LIN {X 0,Y 426.46,Z 439.109,A -85,B 0,C 180,E1 20323.799,E2 20323.799} C_VEL
LIN {X 0,Y 426.439,Z 439.071,A -85,B 0,C 180,E1 20319.981,E2 20319.981} C_VEL
LIN {X 0,Y 426.472,Z 439.347,A -85,B 0,C 180,E1 20317.968,E2 20317.968} C_VEL
LIN {X 0,Y 426.886,Z 440.796,A -85,B 0,C 180,E1 20317.446,E2 20317.446} C_VEL
LIN {X 0,Y 428.773,Z 443.794,A -85,B 0,C 180,E1 20316.644,E2 20316.644} C_VEL
LIN {X 0,Y 432.18,Z 446.15,A -85,B 0,C 180,E1 20315.426,E2 20315.426} C_VEL
LIN {X 0,Y 434.235,Z 449.727,A -85,B 0,C 180,E1 20314.641,E2 20314.641} C_VEL
LIN {X 0,Y 437.693,Z 452.592,A -85,B 0,C 180,E1 20313.51,E2 20313.51} C_VEL
LIN {X 0,Y 440.242,Z 456.382,A -85,B 0,C 180,E1 20312.654,E2 20312.654} C_VEL
LIN {X 0,Y 443.022,Z 458.925,A -85,B 0,C 180,E1 20311.818,E2 20311.818} C_VEL
LIN {X 0,Y 446.073,Z 463.006,A -85,B 0,C 180,E1 20310.895,E2 20310.895} C_VEL
LIN {X 0,Y 448.159,Z 465.113,A -85,B 0,C 180,E1 20310.31,E2 20310.31} C_VEL
LIN {X 0,Y 451.831,Z 469.632,A -85,B 0,C 180,E1 20309.293,E2 20309.293} C_VEL
LIN {X 0,Y 458.066,Z 477.379,A -85,B 0,C 180,E1 20307.67,E2 20307.67} C_VEL
LIN {X 0,Y 466.132,Z 487.643,A -85,B 0,C 180,E1 20305.73,E2 20305.73} C_VEL
LIN {X 0,Y 477.609,Z 503.007,A -85,B 0,C 180,E1 20303.219,E2 20303.219} C_VEL
LIN {X 0,Y 488.82,Z 519.176,A -85,B 0,C 180,E1 20300.986,E2 20300.986} C_VEL
LIN {X 0,Y 501.507,Z 538.911,A -85,B 0,C 180,E1 20298.667,E2 20298.667} C_VEL
LIN {X 0,Y 501.955,Z 540.091,A -85,B 0,C 180,E1 20298.578,E2 20298.578} C_VEL
LIN {X 0,Y 490.454,Z 788.265,A -85,B 0,C 180,E1 20294.759,E2 20294.759} C_VEL
LIN {X 0,Y 488.572,Z 820.608,A -85,B 0,C 180,E1 20294.196,E2 20294.196} C_VEL
LIN {X 0,Y 486.489,Z 842.167,A -85,B 0,C 180,E1 20293.667,E2 20293.667} C_VEL
LIN {X 0,Y 483.443,Z 866.539,A -85,B 0,C 180,E1 20292.88,E2 20292.88} C_VEL
LIN {X 0,Y 480.104,Z 887.806,A -85,B 0,C 180,E1 20292.002,E2 20292.002} C_VEL
LIN {X 0,Y 476.07,Z 910.307,A -85,B 0,C 180,E1 20290.877,E2 20290.877} C_VEL
LIN {X 0,Y 471.559,Z 931.55,A -85,B 0,C 180,E1 20289.582,E2 20289.582} C_VEL
LIN {X 0,Y 467.148,Z 950.701,A -85,B 0,C 180,E1 20288.213,E2 20288.213} C_VEL
LIN {X 0,Y 461.702,Z 972.184,A -85,B 0,C 180,E1 20286.398,E2 20286.398} C_VEL
LIN {X 0,Y 457.123,Z 989.065,A -85,B 0,C 180,E1 20284.737,E2 20284.737} C_VEL
LIN {X 0,Y 451.657,Z 1008.264,A -85,B 0,C 180,E1 20282.545,E2 20282.545} C_VEL
LIN {X 0,Y 447.122,Z 1023.569,A -85,B 0,C 180,E1 20280.507,E2 20280.507} C_VEL
LIN {X 0,Y 442.375,Z 1039.686,A -85,B 0,C 180,E1 20278.043,E2 20278.043} C_VEL
LIN {X 0,Y 438.01,Z 1054.252,A -85,B 0,C 180,E1 20275.415,E2 20275.415} C_VEL
LIN {X 0,Y 434.208,Z 1067.674,A -85,B 0,C 180,E1 20272.617,E2 20272.617} C_VEL
LIN {X 0,Y 430.942,Z 1079.536,A -85,B 0,C 180,E1 20269.66,E2 20269.66} C_VEL
LIN {X 0,Y 428.463,Z 1089.76,A -85,B 0,C 180,E1 20266.681,E2 20266.681} C_VEL
LIN {X 0,Y 426.561,Z 1098.496,A -85,B 0,C 180,E1 20263.557,E2 20263.557} C_VEL
LIN {X 0,Y 425.386,Z 1105.117,A -85,B 0,C 180,E1 20260.702,E2 20260.702} C_VEL
LIN {X 0,Y 424.55,Z 1111.253,A -85,B 0,C 180,E1 20257.307,E2 20257.307} C_VEL
LIN {X 0,Y 424.199,Z 1115.035,A -85,B 0,C 180,E1 20254.461,E2 20254.461} C_VEL
LIN {X 0,Y 424.092,Z 1116.75,A -85,B 0,C 180,E1 20252.744,E2 20252.744} C_VEL
LIN {X 0,Y 423.061,Z 1117.653,A -85,B 0,C 180,E1 20251.71,E2 20251.71} C_VEL
LIN {X 0,Y 416.526,Z 1119.369,A -85,B 0,C 180,E1 20248.791,E2 20248.791} C_VEL
LIN {X 0,Y 415.991,Z 1119.509,A -85,B 0,C 180,E1 20248.026,E2 20248.026} C_VEL
LIN {X 0,Y 415.985,Z 1119.493,A -85,B 0,C 180,E1 20245.312,E2 20245.312} C_VEL
LIN {X 0,Y 416.079,Z 1118.241,A -85,B 0,C 180,E1 20242.127,E2 20242.127} C_VEL
LIN {X 0,Y 416.288,Z 1115.397,A -85,B 0,C 180,E1 20238.921,E2 20238.921} C_VEL
LIN {X 0,Y 416.731,Z 1111.601,A -85,B 0,C 180,E1 20235.975,E2 20235.975} C_VEL
LIN {X 0,Y 417.783,Z 1105.394,A -85,B 0,C 180,E1 20232.449,E2 20232.449} C_VEL
LIN {X 0,Y 419.208,Z 1098.674,A -85,B 0,C 180,E1 20229.474,E2 20229.474} C_VEL
LIN {X 0,Y 421.493,Z 1089.722,A -85,B 0,C 180,E1 20226.216,E2 20226.216} C_VEL
LIN {X 0,Y 424.298,Z 1079.776,A -85,B 0,C 180,E1 20223.249,E2 20223.249} C_VEL
LIN {X 0,Y 427.904,Z 1068.257,A -85,B 0,C 180,E1 20220.305,E2 20220.305} C_VEL
LIN {X 0,Y 432.084,Z 1055.296,A -85,B 0,C 180,E1 20217.529,E2 20217.529} C_VEL
LIN {X 0,Y 436.523,Z 1042.037,A -85,B 0,C 180,E1 20215.065,E2 20215.065} C_VEL
LIN {X 0,Y 441.971,Z 1025.703,A -85,B 0,C 180,E1 20212.47,E2 20212.47} C_VEL
LIN {X 0,Y 446.987,Z 1010.498,A -85,B 0,C 180,E1 20210.392,E2 20210.392} C_VEL
LIN {X 0,Y 453.134,Z 991.205,A -85,B 0,C 180,E1 20208.125,E2 20208.125} C_VEL
LIN {X 0,Y 458.273,Z 974.105,A -85,B 0,C 180,E1 20206.412,E2 20206.412} C_VEL
LIN {X 0,Y 463.989,Z 954.018,A -85,B 0,C 180,E1 20204.671,E2 20204.671} C_VEL
LIN {X 0,Y 469.122,Z 933.798,A -85,B 0,C 180,E1 20203.202,E2 20203.202} C_VEL
LIN {X 0,Y 473.862,Z 913.586,A -85,B 0,C 180,E1 20201.952,E2 20201.952} C_VEL
LIN {X 0,Y 478.549,Z 890.327,A -85,B 0,C 180,E1 20200.763,E2 20200.763} C_VEL
LIN {X 0,Y 482.046,Z 870.182,A -85,B 0,C 180,E1 20199.918,E2 20199.918} C_VEL
LIN {X 0,Y 485.569,Z 845.453,A -85,B 0,C 180,E1 20199.092,E2 20199.092} C_VEL
LIN {X 0,Y 487.926,Z 823.544,A -85,B 0,C 180,E1 20198.542,E2 20198.542} C_VEL
LIN {X 0,Y 489.763,Z 798.161,A -85,B 0,C 180,E1 20198.071,E2 20198.071} C_VEL
LIN {X 0,Y 502.56,Z 550.013,A -85,B 0,C 180,E1 20194.222,E2 20194.222} C_VEL
LIN {X 0,Y 502.637,Z 546.862,A -85,B 0,C 180,E1 20194.158,E2 20194.158} C_VEL
LIN {X 0,Y 491.988,Z 530.606,A -85,B 0,C 180,E1 20191.967,E2 20191.967} C_VEL
LIN {X 0,Y 481.908,Z 516.077,A -85,B 0,C 180,E1 20189.695,E2 20189.695} C_VEL
LIN {X 0,Y 470.549,Z 500.825,A -85,B 0,C 180,E1 20186.843,E2 20186.843} C_VEL
LIN {X 0,Y 464.667,Z 493.605,A -85,B 0,C 180,E1 20185.218,E2 20185.218} C_VEL
LIN {X 0,Y 461.386,Z 489.465,A -85,B 0,C 180,E1 20184.247,E2 20184.247} C_VEL
LIN {X 0,Y 456.943,Z 483.981,A -85,B 0,C 180,E1 20182.856,E2 20182.856} C_VEL
LIN {X 0,Y 453.182,Z 479.216,A -85,B 0,C 180,E1 20181.587,E2 20181.587} C_VEL
LIN {X 0,Y 449.14,Z 474.869,A -85,B 0,C 180,E1 20180.152,E2 20180.152} C_VEL
LIN {X 0,Y 447.664,Z 472.755,A -85,B 0,C 180,E1 20179.575,E2 20179.575} C_VEL
LIN {X 0,Y 444.246,Z 469.377,A -85,B 0,C 180,E1 20178.232,E2 20178.232} C_VEL
LIN {X 0,Y 442.58,Z 466.748,A -85,B 0,C 180,E1 20177.486,E2 20177.486} C_VEL
LIN {X 0,Y 439.326,Z 464.015,A -85,B 0,C 180,E1 20176.053,E2 20176.053} C_VEL
LIN {X 0,Y 437.017,Z 460.34,A -85,B 0,C 180,E1 20174.848,E2 20174.848} C_VEL
LIN {X 0,Y 433.502,Z 457.818,A -85,B 0,C 180,E1 20172.996,E2 20172.996} C_VEL
LIN {X 0,Y 431.27,Z 453.931,A -85,B 0,C 180,E1 20171.501,E2 20171.501} C_VEL
LIN {X 0,Y 427.253,Z 451.254,A -85,B 0,C 180,E1 20168.614,E2 20168.614} C_VEL
LIN {X 0,Y 425.405,Z 447.905,A -85,B 0,C 180,E1 20166.681,E2 20166.681} C_VEL
LIN {X 0,Y 424.103,Z 446.752,A -85,B 0,C 180,E1 20165.14,E2 20165.14} C_VEL
LIN {X 0,Y 421.605,Z 445.43,A -85,B 0,C 180,E1 20158.777,E2 20158.777} C_VEL
LIN {X 0,Y 423.828,Z 446.628,A -85,B 0,C 180,E1 20152.681,E2 20152.681} C_VEL
LIN {X 0,Y 425.295,Z 447.708,A -85,B 0,C 180,E1 20150.912,E2 20150.912} C_VEL
LIN {X 0,Y 427.312,Z 451.295,A -85,B 0,C 180,E1 20148.801,E2 20148.801} C_VEL
LIN {X 0,Y 431.535,Z 454.284,A -85,B 0,C 180,E1 20145.782,E2 20145.782} C_VEL
LIN {X 0,Y 433.596,Z 457.858,A -85,B 0,C 180,E1 20144.416,E2 20144.416} C_VEL
LIN {X 0,Y 437.41,Z 460.857,A -85,B 0,C 180,E1 20142.409,E2 20142.409} C_VEL
LIN {X 0,Y 439.838,Z 464.601,A -85,B 0,C 180,E1 20141.167,E2 20141.167} C_VEL
LIN {X 0,Y 442.831,Z 467.253,A -85,B 0,C 180,E1 20139.859,E2 20139.859} C_VEL
LIN {X 0,Y 448.06,Z 474.081,A -85,B 0,C 180,E1 20137.705,E2 20137.705} C_VEL
LIN {X 0,Y 451.148,Z 477.881,A -85,B 0,C 180,E1 20136.557,E2 20136.557} C_VEL
LIN {X 0,Y 456.118,Z 484.462,A -85,B 0,C 180,E1 20134.831,E2 20134.831} C_VEL
LIN {X 0,Y 462.851,Z 493.629,A -85,B 0,C 180,E1 20132.708,E2 20132.708} C_VEL
LIN {X 0,Y 470.507,Z 504.351,A -85,B 0,C 180,E1 20130.53,E2 20130.53} C_VEL
LIN {X 0,Y 479.766,Z 518.204,A -85,B 0,C 180,E1 20128.143,E2 20128.143} C_VEL
LIN {X 0,Y 489.997,Z 534.394,A -85,B 0,C 180,E1 20125.757,E2 20125.757} C_VEL
LIN {X 0,Y 500.548,Z 552.647,A -85,B 0,C 180,E1 20123.503,E2 20123.503} C_VEL
LIN {X 0,Y 502.46,Z 556.456,A -85,B 0,C 180,E1 20123.105,E2 20123.105} C_VEL
LIN {X 0,Y 491.286,Z 774.343,A -85,B 0,C 180,E1 20119.712,E2 20119.712} C_VEL
LIN {X 0,Y 487.957,Z 837.015,A -85,B 0,C 180,E1 20118.712,E2 20118.712} C_VEL
LIN {X 0,Y 485.355,Z 862.027,A -85,B 0,C 180,E1 20118.161,E2 20118.161} C_VEL
LIN {X 0,Y 482.318,Z 883.724,A -85,B 0,C 180,E1 20117.534,E2 20117.534} C_VEL
LIN {X 0,Y 478.102,Z 908.208,A -85,B 0,C 180,E1 20116.615,E2 20116.615} C_VEL
LIN {X 0,Y 473.961,Z 928.701,A -85,B 0,C 180,E1 20115.657,E2 20115.657} C_VEL
LIN {X 0,Y 468.64,Z 952.137,A -85,B 0,C 180,E1 20114.327,E2 20114.327} C_VEL
LIN {X 0,Y 463.55,Z 971.992,A -85,B 0,C 180,E1 20112.971,E2 20112.971} C_VEL
LIN {X 0,Y 457.782,Z 993.134,A -85,B 0,C 180,E1 20111.272,E2 20111.272} C_VEL
LIN {X 0,Y 452.241,Z 1011.721,A -85,B 0,C 180,E1 20109.499,E2 20109.499} C_VEL
LIN {X 0,Y 446.85,Z 1029.266,A -85,B 0,C 180,E1 20107.572,E2 20107.572} C_VEL
LIN {X 0,Y 440.903,Z 1047.883,A -85,B 0,C 180,E1 20105.172,E2 20105.172} C_VEL
LIN {X 0,Y 436.087,Z 1062.963,A -85,B 0,C 180,E1 20102.916,E2 20102.916} C_VEL
LIN {X 0,Y 430.911,Z 1079.333,A -85,B 0,C 180,E1 20100.058,E2 20100.058} C_VEL
LIN {X 0,Y 427.044,Z 1092.048,A -85,B 0,C 180,E1 20097.469,E2 20097.469} C_VEL
LIN {X 0,Y 423.093,Z 1105.982,A -85,B 0,C 180,E1 20094.133,E2 20094.133} C_VEL
LIN {X 0,Y 420.586,Z 1115.872,A -85,B 0,C 180,E1 20091.33,E2 20091.33} C_VEL
LIN {X 0,Y 418.345,Z 1126.251,A -85,B 0,C 180,E1 20087.814,E2 20087.814} C_VEL
LIN {X 0,Y 417.128,Z 1133.344,A -85,B 0,C 180,E1 20084.862,E2 20084.862} C_VEL
LIN {X 0,Y 416.363,Z 1139.65,A -85,B 0,C 180,E1 20081.638,E2 20081.638} C_VEL
LIN {X 0,Y 416.046,Z 1144.213,A -85,B 0,C 180,E1 20078.43,E2 20078.43} C_VEL
LIN {X 0,Y 415.959,Z 1147.017,A -85,B 0,C 180,E1 20075.656,E2 20075.656} C_VEL
LIN {X 0,Y 415.968,Z 1148.924,A -85,B 0,C 180,E1 20072.48,E2 20072.48} C_VEL
LIN {X 0,Y 415.979,Z 1149.195,A -85,B 0,C 180,E1 20069.404,E2 20069.404} C_VEL
LIN {X 0,Y 415.969,Z 1148.403,A -85,B 0,C 180,E1 20066.831,E2 20066.831} C_VEL
LIN {X 0,Y 415.973,Z 1146.597,A -85,B 0,C 180,E1 20064.206,E2 20064.206} C_VEL
LIN {X 0,Y 416.069,Z 1143.094,A -85,B 0,C 180,E1 20061.01,E2 20061.01} C_VEL
LIN {X 0,Y 416.452,Z 1137.87,A -85,B 0,C 180,E1 20057.802,E2 20057.802} C_VEL
LIN {X 0,Y 417.143,Z 1132.089,A -85,B 0,C 180,E1 20054.997,E2 20054.997} C_VEL
LIN {X 0,Y 418.646,Z 1123.03,A -85,B 0,C 180,E1 20051.477,E2 20051.477} C_VEL
LIN {X 0,Y 420.46,Z 1114.223,A -85,B 0,C 180,E1 20048.663,E2 20048.663} C_VEL
LIN {X 0,Y 423.336,Z 1102.294,A -85,B 0,C 180,E1 20045.436,E2 20045.436} C_VEL
LIN {X 0,Y 426.568,Z 1090.052,A -85,B 0,C 180,E1 20042.649,E2 20042.649} C_VEL
LIN {X 0,Y 430.565,Z 1076.099,A -85,B 0,C 180,E1 20039.893,E2 20039.893} C_VEL
LIN {X 0,Y 435.182,Z 1060.223,A -85,B 0,C 180,E1 20037.24,E2 20037.24} C_VEL
LIN {X 0,Y 440.295,Z 1043.196,A -85,B 0,C 180,E1 20034.772,E2 20034.772} C_VEL
LIN {X 0,Y 445.372,Z 1025.808,A -85,B 0,C 180,E1 20032.632,E2 20032.632} C_VEL
LIN {X 0,Y 450.584,Z 1007.658,A -85,B 0,C 180,E1 20030.687,E2 20030.687} C_VEL
LIN {X 0,Y 456.176,Z 986.891,A -85,B 0,C 180,E1 20028.802,E2 20028.802} C_VEL
LIN {X 0,Y 460.927,Z 968.157,A -85,B 0,C 180,E1 20027.341,E2 20027.341} C_VEL
LIN {X 0,Y 466.322,Z 944.965,A -85,B 0,C 180,E1 20025.824,E2 20025.824} C_VEL
LIN {X 0,Y 470.495,Z 924.844,A -85,B 0,C 180,E1 20024.724,E2 20024.724} C_VEL
LIN {X 0,Y 475.036,Z 899.834,A -85,B 0,C 180,E1 20023.608,E2 20023.608} C_VEL
LIN {X 0,Y 478.393,Z 877.83,A -85,B 0,C 180,E1 20022.836,E2 20022.836} C_VEL
LIN {X 0,Y 481.549,Z 851.869,A -85,B 0,C 180,E1 20022.143,E2 20022.143} C_VEL
LIN {X 0,Y 483.347,Z 829.268,A -85,B 0,C 180,E1 20021.7,E2 20021.7} C_VEL
LIN {X 0,Y 493.938,Z 604.352,A -85,B 0,C 180,E1 20018.193,E2 20018.193} C_VEL
LIN {X 0,Y 496.302,Z 552.568,A -85,B 0,C 180,E1 20017.368,E2 20017.368} C_VEL
LIN {X 0,Y 485.264,Z 532.833,A -85,B 0,C 180,E1 20015.254,E2 20015.254} C_VEL
LIN {X 0,Y 475.654,Z 517.03,A -85,B 0,C 180,E1 20013.275,E2 20013.275} C_VEL
LIN {X 0,Y 465.604,Z 501.38,A -85,B 0,C 180,E1 20011.025,E2 20011.025} C_VEL
LIN {X 0,Y 456.759,Z 488.546,A -85,B 0,C 180,E1 20008.862,E2 20008.862} C_VEL
LIN {X 0,Y 446.922,Z 474.863,A -85,B 0,C 180,E1 20006.187,E2 20006.187} C_VEL
LIN {X 0,Y 441.259,Z 467.655,A -85,B 0,C 180,E1 20004.499,E2 20004.499} C_VEL
LIN {X 0,Y 434.601,Z 459.158,A -85,B 0,C 180,E1 20002.31,E2 20002.31} C_VEL
LIN {X 0,Y 431.388,Z 455.946,A -85,B 0,C 180,E1 20001.198,E2 20001.198} C_VEL
LIN {X 0,Y 429.776,Z 453.269,A -85,B 0,C 180,E1 20000.567,E2 20000.567} C_VEL
LIN {X 0,Y 426.394,Z 450.626,A -85,B 0,C 180,E1 19999.308,E2 19999.308} C_VEL
LIN {X 0,Y 424.043,Z 446.767,A -85,B 0,C 180,E1 19998.277,E2 19998.277} C_VEL
LIN {X 0,Y 420.526,Z 444.455,A -85,B 0,C 180,E1 19996.792,E2 19996.792} C_VEL
LIN {X 0,Y 418.726,Z 441.079,A -85,B 0,C 180,E1 19995.774,E2 19995.774} C_VEL
LIN {X 0,Y 418.542,Z 440.13,A -85,B 0,C 180,E1 19995.094,E2 19995.094} C_VEL
LIN {X 0,Y 418.532,Z 440.092,A -85,B 0,C 180,E1 19991.158,E2 19991.158} C_VEL
LIN {X 0,Y 418.538,Z 440.058,A -85,B 0,C 180,E1 19987.274,E2 19987.274} C_VEL
LIN {X 0,Y 418.532,Z 440.043,A -85,B 0,C 180,E1 19983.424,E2 19983.424} C_VEL
LIN {X 0,Y 418.546,Z 440.076,A -85,B 0,C 180,E1 19979.589,E2 19979.589} C_VEL
LIN {X 0,Y 418.537,Z 440.068,A -85,B 0,C 180,E1 19975.616,E2 19975.616} C_VEL
LIN {X 0,Y 418.535,Z 440.041,A -85,B 0,C 180,E1 19971.759,E2 19971.759} C_VEL
LIN {X 0,Y 418.514,Z 440.068,A -85,B 0,C 180,E1 19968.003,E2 19968.003} C_VEL
LIN {X 0,Y 418.501,Z 440.084,A -85,B 0,C 180,E1 19964.194,E2 19964.194} C_VEL
LIN {X 0,Y 418.566,Z 440.34,A -85,B 0,C 180,E1 19961.083,E2 19961.083} C_VEL
LIN {X 0,Y 418.885,Z 441.719,A -85,B 0,C 180,E1 19960.517,E2 19960.517} C_VEL
LIN {X 0,Y 420.634,Z 444.556,A -85,B 0,C 180,E1 19959.62,E2 19959.62} C_VEL
LIN {X 0,Y 424.541,Z 447.376,A -85,B 0,C 180,E1 19957.971,E2 19957.971} C_VEL
LIN {X 0,Y 426.527,Z 450.821,A -85,B 0,C 180,E1 19957.098,E2 19957.098} C_VEL
LIN {X 0,Y 429.581,Z 453.153,A -85,B 0,C 180,E1 19955.963,E2 19955.963} C_VEL
LIN {X 0,Y 430.325,Z 454.138,A -85,B 0,C 180,E1 19955.679,E2 19955.679} C_VEL
LIN {X 0,Y 432.755,Z 457.679,A -85,B 0,C 180,E1 19954.767,E2 19954.767} C_VEL
LIN {X 0,Y 435.613,Z 460.182,A -85,B 0,C 180,E1 19953.814,E2 19953.814} C_VEL
LIN {X 0,Y 438.633,Z 464.237,A -85,B 0,C 180,E1 19952.803,E2 19952.803} C_VEL
LIN {X 0,Y 440.788,Z 466.318,A -85,B 0,C 180,E1 19952.141,E2 19952.141} C_VEL
LIN {X 0,Y 444.326,Z 470.77,A -85,B 0,C 180,E1 19951.064,E2 19951.064} C_VEL
LIN {X 0,Y 446.059,Z 472.796,A -85,B 0,C 180,E1 19950.562,E2 19950.562} C_VEL
LIN {X 0,Y 450.981,Z 478.829,A -85,B 0,C 180,E1 19949.192,E2 19949.192} C_VEL
LIN {X 0,Y 456.103,Z 485.324,A -85,B 0,C 180,E1 19947.848,E2 19947.848} C_VEL
LIN {X 0,Y 463.181,Z 494.394,A -85,B 0,C 180,E1 19946.117,E2 19946.117} C_VEL
LIN {X 0,Y 474.648,Z 509.946,A -85,B 0,C 180,E1 19943.554,E2 19943.554} C_VEL
LIN {X 0,Y 485.547,Z 525.916,A -85,B 0,C 180,E1 19941.336,E2 19941.336} C_VEL
LIN {X 0,Y 496.73,Z 543.494,A -85,B 0,C 180,E1 19939.24,E2 19939.24} C_VEL
LIN {X 0,Y 484.803,Z 792.502,A -85,B 0,C 180,E1 19935.383,E2 19935.383} C_VEL
LIN {X 0,Y 482.96,Z 821.822,A -85,B 0,C 180,E1 19934.857,E2 19934.857} C_VEL
LIN {X 0,Y 480.821,Z 843.2,A -85,B 0,C 180,E1 19934.325,E2 19934.325} C_VEL
LIN {X 0,Y 477.432,Z 868.992,A -85,B 0,C 180,E1 19933.471,E2 19933.471} C_VEL
LIN {X 0,Y 474.057,Z 889.712,A -85,B 0,C 180,E1 19932.598,E2 19932.598} C_VEL
LIN {X 0,Y 469.603,Z 913.272,A -85,B 0,C 180,E1 19931.386,E2 19931.386} C_VEL
LIN {X 0,Y 465.228,Z 933.159,A -85,B 0,C 180,E1 19930.149,E2 19930.149} C_VEL
LIN {X 0,Y 460.321,Z 953.773,A -85,B 0,C 180,E1 19928.645,E2 19928.645} C_VEL
LIN {X 0,Y 455.08,Z 973.456,A -85,B 0,C 180,E1 19926.937,E2 19926.937} C_VEL
LIN {X 0,Y 450.365,Z 990.25,A -85,B 0,C 180,E1 19925.257,E2 19925.257} C_VEL
LIN {X 0,Y 444.542,Z 1009.868,A -85,B 0,C 180,E1 19922.968,E2 19922.968} C_VEL
LIN {X 0,Y 439.898,Z 1024.996,A -85,B 0,C 180,E1 19920.911,E2 19920.911} C_VEL
LIN {X 0,Y 434.659,Z 1041.964,A -85,B 0,C 180,E1 19918.23,E2 19918.23} C_VEL
LIN {X 0,Y 430.493,Z 1055.403,A -85,B 0,C 180,E1 19915.743,E2 19915.743} C_VEL
LIN {X 0,Y 426.386,Z 1069.23,A -85,B 0,C 180,E1 19912.764,E2 19912.764} C_VEL
LIN {X 0,Y 423.316,Z 1079.957,A -85,B 0,C 180,E1 19910.029,E2 19910.029} C_VEL
LIN {X 0,Y 420.717,Z 1090.164,A -85,B 0,C 180,E1 19906.997,E2 19906.997} C_VEL
LIN {X 0,Y 418.715,Z 1098.875,A -85,B 0,C 180,E1 19903.816,E2 19903.816} C_VEL
LIN {X 0,Y 417.466,Z 1105.533,A -85,B 0,C 180,E1 19900.884,E2 19900.884} C_VEL
LIN {X 0,Y 416.586,Z 1111.593,A -85,B 0,C 180,E1 19897.447,E2 19897.447} C_VEL
LIN {X 0,Y 416.216,Z 1115.361,A -85,B 0,C 180,E1 19894.547,E2 19894.547} C_VEL
LIN {X 0,Y 416.027,Z 1118.287,A -85,B 0,C 180,E1 19891.239,E2 19891.239} C_VEL
LIN {X 0,Y 415.991,Z 1119.502,A -85,B 0,C 180,E1 19888.072,E2 19888.072} C_VEL
LIN {X 0,Y 415.991,Z 1119.509,A -85,B 0,C 180,E1 19888.026,E2 19888.026} C_VEL
LIN {X 0,Y 415.009,Z 1119.736,A -85,B 0,C 180,E1 19886.965,E2 19886.965} C_VEL
LIN {X 0,Y 408.577,Z 1119.451,A -85,B 0,C 180,E1 19883.975,E2 19883.975} C_VEL
LIN {X 0,Y 408.034,Z 1119.09,A -85,B 0,C 180,E1 19883.196,E2 19883.196} C_VEL
LIN {X 0,Y 408.156,Z 1117.287,A -85,B 0,C 180,E1 19880.411,E2 19880.411} C_VEL
LIN {X 0,Y 408.589,Z 1113.451,A -85,B 0,C 180,E1 19876.845,E2 19876.845} C_VEL
LIN {X 0,Y 409.323,Z 1108.812,A -85,B 0,C 180,E1 19873.831,E2 19873.831} C_VEL
LIN {X 0,Y 410.725,Z 1102.108,A -85,B 0,C 180,E1 19870.414,E2 19870.414} C_VEL
LIN {X 0,Y 412.729,Z 1093.989,A -85,B 0,C 180,E1 19867.193,E2 19867.193} C_VEL
LIN {X 0,Y 415.366,Z 1084.91,A -85,B 0,C 180,E1 19864.169,E2 19864.169} C_VEL
LIN {X 0,Y 418.955,Z 1073.52,A -85,B 0,C 180,E1 19861.021,E2 19861.021} C_VEL
LIN {X 0,Y 422.775,Z 1062.109,A -85,B 0,C 180,E1 19858.329,E2 19858.329} C_VEL
LIN {X 0,Y 428.108,Z 1046.738,A -85,B 0,C 180,E1 19855.257,E2 19855.257} C_VEL
LIN {X 0,Y 432.884,Z 1033.061,A -85,B 0,C 180,E1 19852.924,E2 19852.924} C_VEL
LIN {X 0,Y 438.969,Z 1015.438,A -85,B 0,C 180,E1 19850.345,E2 19850.345} C_VEL
LIN {X 0,Y 444.337,Z 999.378,A -85,B 0,C 180,E1 19848.34,E2 19848.34} C_VEL
LIN {X 0,Y 450.441,Z 980.418,A -85,B 0,C 180,E1 19846.297,E2 19846.297} C_VEL
LIN {X 0,Y 455.879,Z 962.101,A -85,B 0,C 180,E1 19844.624,E2 19844.624} C_VEL
LIN {X 0,Y 461.101,Z 943.313,A -85,B 0,C 180,E1 19843.139,E2 19843.139} C_VEL
LIN {X 0,Y 466.575,Z 921.361,A -85,B 0,C 180,E1 19841.681,E2 19841.681} C_VEL
LIN {X 0,Y 470.861,Z 902.128,A -85,B 0,C 180,E1 19840.609,E2 19840.609} C_VEL
LIN {X 0,Y 475.391,Z 878.698,A -85,B 0,C 180,E1 19839.521,E2 19839.521} C_VEL
LIN {X 0,Y 478.772,Z 857.301,A -85,B 0,C 180,E1 19838.73,E2 19838.73} C_VEL
LIN {X 0,Y 481.845,Z 833.683,A -85,B 0,C 180,E1 19838.04,E2 19838.04} C_VEL
LIN {X 0,Y 483.974,Z 809.348,A -85,B 0,C 180,E1 19837.53,E2 19837.53} C_VEL
LIN {X 0,Y 496.518,Z 575.381,A -85,B 0,C 180,E1 19833.865,E2 19833.865} C_VEL
LIN {X 0,Y 497.779,Z 550.89,A -85,B 0,C 180,E1 19833.469,E2 19833.469} C_VEL
LIN {X 0,Y 486.39,Z 533.438,A -85,B 0,C 180,E1 19831.029,E2 19831.029} C_VEL
LIN {X 0,Y 477.111,Z 520.336,A -85,B 0,C 180,E1 19828.852,E2 19828.852} C_VEL
LIN {X 0,Y 467.91,Z 507.726,A -85,B 0,C 180,E1 19826.459,E2 19826.459} C_VEL
LIN {X 0,Y 459.463,Z 497.013,A -85,B 0,C 180,E1 19824.014,E2 19824.014} C_VEL
LIN {X 0,Y 454.702,Z 491.162,A -85,B 0,C 180,E1 19822.497,E2 19822.497} C_VEL
LIN {X 0,Y 450.397,Z 485.874,A -85,B 0,C 180,E1 19821.01,E2 19821.01} C_VEL
LIN {X 0,Y 446.739,Z 481.525,A -85,B 0,C 180,E1 19819.651,E2 19819.651} C_VEL
LIN {X 0,Y 445.574,Z 480.089,A -85,B 0,C 180,E1 19819.193,E2 19819.193} C_VEL
LIN {X 0,Y 442.111,Z 476.312,A -85,B 0,C 180,E1 19817.778,E2 19817.778} C_VEL
LIN {X 0,Y 440.736,Z 474.286,A -85,B 0,C 180,E1 19817.153,E2 19817.153} C_VEL
LIN {X 0,Y 437.441,Z 471.214,A -85,B 0,C 180,E1 19815.648,E2 19815.648} C_VEL
LIN {X 0,Y 435.543,Z 468.086,A -85,B 0,C 180,E1 19814.627,E2 19814.627} C_VEL
LIN {X 0,Y 432.091,Z 465.501,A -85,B 0,C 180,E1 19812.768,E2 19812.768} C_VEL
LIN {X 0,Y 429.898,Z 461.671,A -85,B 0,C 180,E1 19811.267,E2 19811.267} C_VEL
LIN {X 0,Y 426.124,Z 459.141,A -85,B 0,C 180,E1 19808.501,E2 19808.501} C_VEL
LIN {X 0,Y 424.242,Z 455.75,A -85,B 0,C 180,E1 19806.496,E2 19806.496} C_VEL
LIN {X 0,Y 423.024,Z 454.66,A -85,B 0,C 180,E1 19805.017,E2 19805.017} C_VEL
LIN {X 0,Y 420.63,Z 453.371,A -85,B 0,C 180,E1 19798.774,E2 19798.774} C_VEL
LIN {X 0,Y 422.86,Z 454.575,A -85,B 0,C 180,E1 19792.664,E2 19792.664} C_VEL
LIN {X 0,Y 424.236,Z 455.676,A -85,B 0,C 180,E1 19790.983,E2 19790.983} C_VEL
LIN {X 0,Y 426.039,Z 459.015,A -85,B 0,C 180,E1 19789.041,E2 19789.041} C_VEL
LIN {X 0,Y 429.781,Z 461.587,A -85,B 0,C 180,E1 19786.272,E2 19786.272} C_VEL
LIN {X 0,Y 432.63,Z 466.024,A -85,B 0,C 180,E1 19784.38,E2 19784.38} C_VEL
LIN {X 0,Y 435.825,Z 468.515,A -85,B 0,C 180,E1 19782.682,E2 19782.682} C_VEL
LIN {X 0,Y 438.474,Z 472.437,A -85,B 0,C 180,E1 19781.313,E2 19781.313} C_VEL
LIN {X 0,Y 441.286,Z 475.021,A -85,B 0,C 180,E1 19780.061,E2 19780.061} C_VEL
LIN {X 0,Y 448.943,Z 484.904,A -85,B 0,C 180,E1 19776.956,E2 19776.956} C_VEL
LIN {X 0,Y 454.156,Z 491.981,A -85,B 0,C 180,E1 19775.102,E2 19775.102} C_VEL
LIN {X 0,Y 460.626,Z 500.936,A -85,B 0,C 180,E1 19773.02,E2 19773.02} C_VEL
LIN {X 0,Y 468.796,Z 512.579,A -85,B 0,C 180,E1 19770.657,E2 19770.657} C_VEL
LIN {X 0,Y 479.429,Z 528.801,A -85,B 0,C 180,E1 19767.906,E2 19767.906} C_VEL
LIN {X 0,Y 489.486,Z 545.494,A -85,B 0,C 180,E1 19765.557,E2 19765.557} C_VEL
LIN {X 0,Y 497.614,Z 560.041,A -85,B 0,C 180,E1 19763.799,E2 19763.799} C_VEL
LIN {X 0,Y 486.071,Z 777.932,A -85,B 0,C 180,E1 19760.388,E2 19760.388} C_VEL
LIN {X 0,Y 482.807,Z 837.069,A -85,B 0,C 180,E1 19759.438,E2 19759.438} C_VEL
LIN {X 0,Y 480.136,Z 861.939,A -85,B 0,C 180,E1 19758.886,E2 19758.886} C_VEL
LIN {X 0,Y 476.977,Z 883.884,A -85,B 0,C 180,E1 19758.249,E2 19758.249} C_VEL
LIN {X 0,Y 472.616,Z 908.39,A -85,B 0,C 180,E1 19757.324,E2 19757.324} C_VEL
LIN {X 0,Y 468.36,Z 928.824,A -85,B 0,C 180,E1 19756.363,E2 19756.363} C_VEL
LIN {X 0,Y 462.878,Z 952.174,A -85,B 0,C 180,E1 19755.028,E2 19755.028} C_VEL
LIN {X 0,Y 457.728,Z 971.632,A -85,B 0,C 180,E1 19753.692,E2 19753.692} C_VEL
LIN {X 0,Y 451.88,Z 992.414,A -85,B 0,C 180,E1 19752.017,E2 19752.017} C_VEL
LIN {X 0,Y 445.875,Z 1011.878,A -85,B 0,C 180,E1 19750.146,E2 19750.146} C_VEL
LIN {X 0,Y 440.188,Z 1029.73,A -85,B 0,C 180,E1 19748.16,E2 19748.16} C_VEL
LIN {X 0,Y 434.184,Z 1047.755,A -85,B 0,C 180,E1 19745.799,E2 19745.799} C_VEL
LIN {X 0,Y 428.887,Z 1063.669,A -85,B 0,C 180,E1 19743.381,E2 19743.381} C_VEL
LIN {X 0,Y 423.793,Z 1079.06,A -85,B 0,C 180,E1 19740.639,E2 19740.639} C_VEL
LIN {X 0,Y 419.702,Z 1091.864,A -85,B 0,C 180,E1 19737.991,E2 19737.991} C_VEL
LIN {X 0,Y 415.551,Z 1105.776,A -85,B 0,C 180,E1 19734.599,E2 19734.599} C_VEL
LIN {X 0,Y 412.899,Z 1115.656,A -85,B 0,C 180,E1 19731.747,E2 19731.747} C_VEL
LIN {X 0,Y 410.521,Z 1126.017,A -85,B 0,C 180,E1 19728.166,E2 19728.166} C_VEL
LIN {X 0,Y 409.223,Z 1133.103,A -85,B 0,C 180,E1 19725.156,E2 19725.156} C_VEL
LIN {X 0,Y 408.398,Z 1139.396,A -85,B 0,C 180,E1 19721.868,E2 19721.868} C_VEL
LIN {X 0,Y 408.054,Z 1143.95,A -85,B 0,C 180,E1 19718.596,E2 19718.596} C_VEL
LIN {X 0,Y 407.966,Z 1146.749,A -85,B 0,C 180,E1 19715.767,E2 19715.767} C_VEL
LIN {X 0,Y 407.971,Z 1148.645,A -85,B 0,C 180,E1 19712.528,E2 19712.528} C_VEL
LIN {X 0,Y 407.985,Z 1148.898,A -85,B 0,C 180,E1 19709.337,E2 19709.337} C_VEL
LIN {X 0,Y 407.978,Z 1148.037,A -85,B 0,C 180,E1 19706.628,E2 19706.628} C_VEL
LIN {X 0,Y 407.988,Z 1145.942,A -85,B 0,C 180,E1 19703.668,E2 19703.668} C_VEL
LIN {X 0,Y 408.136,Z 1141.932,A -85,B 0,C 180,E1 19700.268,E2 19700.268} C_VEL
LIN {X 0,Y 408.558,Z 1137.015,A -85,B 0,C 180,E1 19697.275,E2 19697.275} C_VEL
LIN {X 0,Y 409.502,Z 1130.174,A -85,B 0,C 180,E1 19693.983,E2 19693.983} C_VEL
LIN {X 0,Y 411.085,Z 1121.426,A -85,B 0,C 180,E1 19690.683,E2 19690.683} C_VEL
LIN {X 0,Y 413.333,Z 1111.496,A -85,B 0,C 180,E1 19687.529,E2 19687.529} C_VEL
LIN {X 0,Y 416.4,Z 1099.549,A -85,B 0,C 180,E1 19684.391,E2 19684.391} C_VEL
LIN {X 0,Y 419.972,Z 1087.045,A -85,B 0,C 180,E1 19681.564,E2 19681.564} C_VEL
LIN {X 0,Y 424.299,Z 1072.517,A -85,B 0,C 180,E1 19678.772,E2 19678.772} C_VEL
LIN {X 0,Y 428.753,Z 1058.04,A -85,B 0,C 180,E1 19676.363,E2 19676.363} C_VEL
LIN {X 0,Y 434.459,Z 1039.619,A -85,B 0,C 180,E1 19673.738,E2 19673.738} C_VEL
LIN {X 0,Y 439.377,Z 1023.431,A -85,B 0,C 180,E1 19671.757,E2 19671.757} C_VEL
LIN {X 0,Y 445.321,Z 1003.183,A -85,B 0,C 180,E1 19669.626,E2 19669.626} C_VEL
LIN {X 0,Y 450.402,Z 984.835,A -85,B 0,C 180,E1 19667.984,E2 19667.984} C_VEL
LIN {X 0,Y 455.874,Z 963.878,A -85,B 0,C 180,E1 19666.37,E2 19666.37} C_VEL
LIN {X 0,Y 460.94,Z 942.268,A -85,B 0,C 180,E1 19664.994,E2 19664.994} C_VEL
LIN {X 0,Y 465.595,Z 920.305,A -85,B 0,C 180,E1 19663.815,E2 19663.815} C_VEL
LIN {X 0,Y 469.713,Z 897.509,A -85,B 0,C 180,E1 19662.832,E2 19662.832} C_VEL
LIN {X 0,Y 473.087,Z 875.77,A -85,B 0,C 180,E1 19662.08,E2 19662.08} C_VEL
LIN {X 0,Y 476.23,Z 849.82,A -85,B 0,C 180,E1 19661.403,E2 19661.403} C_VEL
LIN {X 0,Y 478.004,Z 827.39,A -85,B 0,C 180,E1 19660.968,E2 19660.968} C_VEL
LIN {X 0,Y 488.95,Z 602.172,A -85,B 0,C 180,E1 19657.436,E2 19657.436} C_VEL
LIN {X 0,Y 491.115,Z 556.093,A -85,B 0,C 180,E1 19656.695,E2 19656.695} C_VEL
LIN {X 0,Y 480.584,Z 537.168,A -85,B 0,C 180,E1 19654.611,E2 19654.611} C_VEL
LIN {X 0,Y 469.777,Z 519.215,A -85,B 0,C 180,E1 19652.292,E2 19652.292} C_VEL
LIN {X 0,Y 458.2,Z 501.404,A -85,B 0,C 180,E1 19649.55,E2 19649.55} C_VEL
LIN {X 0,Y 447.654,Z 486.414,A -85,B 0,C 180,E1 19646.749,E2 19646.749} C_VEL
LIN {X 0,Y 442.891,Z 480.104,A -85,B 0,C 180,E1 19645.365,E2 19645.365} C_VEL
LIN {X 0,Y 439.123,Z 475.014,A -85,B 0,C 180,E1 19644.196,E2 19644.196} C_VEL
LIN {X 0,Y 432.547,Z 466.571,A -85,B 0,C 180,E1 19641.993,E2 19641.993} C_VEL
LIN {X 0,Y 429.22,Z 463.073,A -85,B 0,C 180,E1 19640.809,E2 19640.809} C_VEL
LIN {X 0,Y 427.784,Z 460.77,A -85,B 0,C 180,E1 19640.239,E2 19640.239} C_VEL
LIN {X 0,Y 424.474,Z 457.977,A -85,B 0,C 180,E1 19638.97,E2 19638.97} C_VEL
LIN {X 0,Y 422.46,Z 454.5,A -85,B 0,C 180,E1 19638.063,E2 19638.063} C_VEL
LIN {X 0,Y 418.99,Z 452.142,A -85,B 0,C 180,E1 19636.57,E2 19636.57} C_VEL
LIN {X 0,Y 417.008,Z 448.893,A -85,B 0,C 180,E1 19635.542,E2 19635.542} C_VEL
LIN {X 0,Y 416.049,Z 447.727,A -85,B 0,C 180,E1 19635.044,E2 19635.044} C_VEL
LIN {X 0,Y 412.517,Z 445.326,A -85,B 0,C 180,E1 19633.17,E2 19633.17} C_VEL
LIN {X 0,Y 410.736,Z 441.861,A -85,B 0,C 180,E1 19631.8,E2 19631.8} C_VEL
LIN {X 0,Y 410.594,Z 441.11,A -85,B 0,C 180,E1 19630.808,E2 19630.808} C_VEL
LIN {X 0,Y 410.583,Z 441.057,A -85,B 0,C 180,E1 19626.853,E2 19626.853} C_VEL
LIN {X 0,Y 410.578,Z 441.032,A -85,B 0,C 180,E1 19622.931,E2 19622.931} C_VEL
LIN {X 0,Y 410.586,Z 441.049,A -85,B 0,C 180,E1 19619.023,E2 19619.023} C_VEL
LIN {X 0,Y 410.587,Z 441.073,A -85,B 0,C 180,E1 19615.11,E2 19615.11} C_VEL
LIN {X 0,Y 410.595,Z 441.031,A -85,B 0,C 180,E1 19611.316,E2 19611.316} C_VEL
LIN {X 0,Y 410.598,Z 441.041,A -85,B 0,C 180,E1 19607.483,E2 19607.483} C_VEL
LIN {X 0,Y 410.631,Z 441.367,A -85,B 0,C 180,E1 19605.042,E2 19605.042} C_VEL
LIN {X 0,Y 410.999,Z 442.865,A -85,B 0,C 180,E1 19604.297,E2 19604.297} C_VEL
LIN {X 0,Y 412.949,Z 445.817,A -85,B 0,C 180,E1 19603.036,E2 19603.036} C_VEL
LIN {X 0,Y 416.747,Z 448.37,A -85,B 0,C 180,E1 19601.064,E2 19601.064} C_VEL
LIN {X 0,Y 418.697,Z 451.802,A -85,B 0,C 180,E1 19600.032,E2 19600.032} C_VEL
LIN {X 0,Y 421.963,Z 454.319,A -85,B 0,C 180,E1 19598.597,E2 19598.597} C_VEL
LIN {X 0,Y 422.724,Z 455.05,A -85,B 0,C 180,E1 19598.273,E2 19598.273} C_VEL
LIN {X 0,Y 425.094,Z 458.73,A -85,B 0,C 180,E1 19597.236,E2 19597.236} C_VEL
LIN {X 0,Y 428.189,Z 461.349,A -85,B 0,C 180,E1 19596.063,E2 19596.063} C_VEL
LIN {X 0,Y 430.927,Z 465.236,A -85,B 0,C 180,E1 19595.02,E2 19595.02} C_VEL
LIN {X 0,Y 433.555,Z 467.689,A -85,B 0,C 180,E1 19594.122,E2 19594.122} C_VEL
LIN {X 0,Y 436.934,Z 471.976,A -85,B 0,C 180,E1 19592.983,E2 19592.983} C_VEL
LIN {X 0,Y 438.664,Z 473.82,A -85,B 0,C 180,E1 19592.437,E2 19592.437} C_VEL
LIN {X 0,Y 442.379,Z 478.331,A -85,B 0,C 180,E1 19591.295,E2 19591.295} C_VEL
LIN {X 0,Y 448.64,Z 486.164,A -85,B 0,C 180,E1 19589.496,E2 19589.496} C_VEL
LIN {X 0,Y 455.943,Z 495.394,A -85,B 0,C 180,E1 19587.575,E2 19587.575} C_VEL
LIN {X 0,Y 467.078,Z 510.429,A -85,B 0,C 180,E1 19584.915,E2 19584.915} C_VEL
LIN {X 0,Y 477.442,Z 525.245,A -85,B 0,C 180,E1 19582.678,E2 19582.678} C_VEL
LIN {X 0,Y 490.507,Z 545.523,A -85,B 0,C 180,E1 19580.107,E2 19580.107} C_VEL
LIN {X 0,Y 491.531,Z 547.642,A -85,B 0,C 180,E1 19579.904,E2 19579.904} C_VEL
LIN {X 0,Y 479.167,Z 797.647,A -85,B 0,C 180,E1 19576.007,E2 19576.007} C_VEL
LIN {X 0,Y 477.401,Z 823.191,A -85,B 0,C 180,E1 19575.53,E2 19575.53} C_VEL
LIN {X 0,Y 475.151,Z 844.871,A -85,B 0,C 180,E1 19574.981,E2 19574.981} C_VEL
LIN {X 0,Y 471.703,Z 869.989,A -85,B 0,C 180,E1 19574.134,E2 19574.134} C_VEL
LIN {X 0,Y 468.28,Z 890.361,A -85,B 0,C 180,E1 19573.268,E2 19573.268} C_VEL
LIN {X 0,Y 463.651,Z 914.042,A -85,B 0,C 180,E1 19572.037,E2 19572.037} C_VEL
LIN {X 0,Y 459.148,Z 933.879,A -85,B 0,C 180,E1 19570.792,E2 19570.792} C_VEL
LIN {X 0,Y 453.892,Z 955.181,A -85,B 0,C 180,E1 19569.216,E2 19569.216} C_VEL
LIN {X 0,Y 448.499,Z 974.725,A -85,B 0,C 180,E1 19567.491,E2 19567.491} C_VEL
LIN {X 0,Y 443.13,Z 993.224,A -85,B 0,C 180,E1 19565.603,E2 19565.603} C_VEL
LIN {X 0,Y 437.497,Z 1011.33,A -85,B 0,C 180,E1 19563.422,E2 19563.422} C_VEL
LIN {X 0,Y 432.696,Z 1026.421,A -85,B 0,C 180,E1 19561.328,E2 19561.328} C_VEL
LIN {X 0,Y 427.381,Z 1042.911,A -85,B 0,C 180,E1 19558.66,E2 19558.66} C_VEL
LIN {X 0,Y 423.204,Z 1055.869,A -85,B 0,C 180,E1 19556.22,E2 19556.22} C_VEL
LIN {X 0,Y 418.914,Z 1069.664,A -85,B 0,C 180,E1 19553.193,E2 19553.193} C_VEL
LIN {X 0,Y 415.711,Z 1080.376,A -85,B 0,C 180,E1 19550.412,E2 19550.412} C_VEL
LIN {X 0,Y 412.984,Z 1090.564,A -85,B 0,C 180,E1 19547.326,E2 19547.326} C_VEL
LIN {X 0,Y 410.878,Z 1099.253,A -85,B 0,C 180,E1 19544.085,E2 19544.085} C_VEL
LIN {X 0,Y 409.541,Z 1106.01,A -85,B 0,C 180,E1 19541.042,E2 19541.042} C_VEL
LIN {X 0,Y 408.625,Z 1111.932,A -85,B 0,C 180,E1 19537.593,E2 19537.593} C_VEL
LIN {X 0,Y 408.245,Z 1115.532,A -85,B 0,C 180,E1 19534.777,E2 19534.777} C_VEL
LIN {X 0,Y 408.05,Z 1118.41,A -85,B 0,C 180,E1 19531.545,E2 19531.545} C_VEL
LIN {X 0,Y 407.99,Z 1119.748,A -85,B 0,C 180,E1 19528.315,E2 19528.315} C_VEL
LIN {X 0,Y 407.992,Z 1119.815,A -85,B 0,C 180,E1 19525.502,E2 19525.502} C_VEL
LIN {X 0,Y 408.034,Z 1119.09,A -85,B 0,C 180,E1 19523.196,E2 19523.196} C_VEL
LIN {X 0,Y 407.048,Z 1118.635,A -85,B 0,C 180,E1 19522.116,E2 19522.116} C_VEL
LIN {X 0,Y 400.827,Z 1116.525,A -85,B 0,C 180,E1 19519.076,E2 19519.076} C_VEL
LIN {X 0,Y 400.385,Z 1115.692,A -85,B 0,C 180,E1 19518.288,E2 19518.288} C_VEL
LIN {X 0,Y 401.019,Z 1111.469,A -85,B 0,C 180,E1 19514.971,E2 19514.971} C_VEL
LIN {X 0,Y 402.253,Z 1105.226,A -85,B 0,C 180,E1 19511.447,E2 19511.447} C_VEL
LIN {X 0,Y 403.953,Z 1098.383,A -85,B 0,C 180,E1 19508.357,E2 19508.357} C_VEL
LIN {X 0,Y 406.734,Z 1088.713,A -85,B 0,C 180,E1 19504.831,E2 19504.831} C_VEL
LIN {X 0,Y 409.836,Z 1079.081,A -85,B 0,C 180,E1 19501.909,E2 19501.909} C_VEL
LIN {X 0,Y 414.361,Z 1066.025,A -85,B 0,C 180,E1 19498.585,E2 19498.585} C_VEL
LIN {X 0,Y 418.75,Z 1053.802,A -85,B 0,C 180,E1 19495.952,E2 19495.952} C_VEL
LIN {X 0,Y 424.458,Z 1038.198,A -85,B 0,C 180,E1 19493.08,E2 19493.08} C_VEL
LIN {X 0,Y 429.734,Z 1023.574,A -85,B 0,C 180,E1 19490.788,E2 19490.788} C_VEL
LIN {X 0,Y 435.813,Z 1006.483,A -85,B 0,C 180,E1 19488.466,E2 19488.466} C_VEL
LIN {X 0,Y 441.943,Z 988.137,A -85,B 0,C 180,E1 19486.365,E2 19486.365} C_VEL
LIN {X 0,Y 448.196,Z 968.654,A -85,B 0,C 180,E1 19484.447,E2 19484.447} C_VEL
LIN {X 0,Y 453.919,Z 948.905,A -85,B 0,C 180,E1 19482.816,E2 19482.816} C_VEL
LIN {X 0,Y 459.016,Z 929.87,A -85,B 0,C 180,E1 19481.466,E2 19481.466} C_VEL
LIN {X 0,Y 464.351,Z 907.552,A -85,B 0,C 180,E1 19480.144,E2 19480.144} C_VEL
LIN {X 0,Y 468.684,Z 886.509,A -85,B 0,C 180,E1 19479.109,E2 19479.109} C_VEL
LIN {X 0,Y 473.077,Z 861.122,A -85,B 0,C 180,E1 19478.108,E2 19478.108} C_VEL
LIN {X 0,Y 476.055,Z 839.391,A -85,B 0,C 180,E1 19477.444,E2 19477.444} C_VEL
LIN {X 0,Y 478.673,Z 813.636,A -85,B 0,C 180,E1 19476.86,E2 19476.86} C_VEL
LIN {X 0,Y 483.736,Z 723.149,A -85,B 0,C 180,E1 19475.417,E2 19475.417} C_VEL
LIN {X 0,Y 493.064,Z 555.091,A -85,B 0,C 180,E1 19472.783,E2 19472.783} C_VEL
LIN {X 0,Y 482.041,Z 538.119,A -85,B 0,C 180,E1 19470.337,E2 19470.337} C_VEL
LIN {X 0,Y 472.01,Z 523.852,A -85,B 0,C 180,E1 19467.881,E2 19467.881} C_VEL
LIN {X 0,Y 464.281,Z 513.405,A -85,B 0,C 180,E1 19465.788,E2 19465.788} C_VEL
LIN {X 0,Y 457.357,Z 504.365,A -85,B 0,C 180,E1 19463.72,E2 19463.72} C_VEL
LIN {X 0,Y 452.303,Z 498.146,A -85,B 0,C 180,E1 19462.075,E2 19462.075} C_VEL
LIN {X 0,Y 448.245,Z 493.104,A -85,B 0,C 180,E1 19460.637,E2 19460.637} C_VEL
LIN {X 0,Y 444.522,Z 488.408,A -85,B 0,C 180,E1 19459.206,E2 19459.206} C_VEL
LIN {X 0,Y 440.275,Z 483.665,A -85,B 0,C 180,E1 19457.444,E2 19457.444} C_VEL
LIN {X 0,Y 439.201,Z 481.988,A -85,B 0,C 180,E1 19456.942,E2 19456.942} C_VEL
LIN {X 0,Y 435.824,Z 478.75,A -85,B 0,C 180,E1 19455.366,E2 19455.366} C_VEL
LIN {X 0,Y 433.821,Z 475.693,A -85,B 0,C 180,E1 19454.278,E2 19454.278} C_VEL
LIN {X 0,Y 430.481,Z 472.917,A -85,B 0,C 180,E1 19452.407,E2 19452.407} C_VEL
LIN {X 0,Y 428.529,Z 469.443,A -85,B 0,C 180,E1 19451.031,E2 19451.031} C_VEL
LIN {X 0,Y 424.997,Z 467.026,A -85,B 0,C 180,E1 19448.388,E2 19448.388} C_VEL
LIN {X 0,Y 423.037,Z 463.438,A -85,B 0,C 180,E1 19446.242,E2 19446.242} C_VEL
LIN {X 0,Y 421.553,Z 462.42,A -85,B 0,C 180,E1 19444.353,E2 19444.353} C_VEL
LIN {X 0,Y 419.659,Z 461.301,A -85,B 0,C 180,E1 19438.498,E2 19438.498} C_VEL
LIN {X 0,Y 422.424,Z 462.763,A -85,B 0,C 180,E1 19431.972,E2 19431.972} C_VEL
LIN {X 0,Y 423.233,Z 463.94,A -85,B 0,C 180,E1 19430.961,E2 19430.961} C_VEL
LIN {X 0,Y 425.219,Z 467.232,A -85,B 0,C 180,E1 19428.883,E2 19428.883} C_VEL
LIN {X 0,Y 428.752,Z 469.76,A -85,B 0,C 180,E1 19426.273,E2 19426.273} C_VEL
LIN {X 0,Y 431.008,Z 473.486,A -85,B 0,C 180,E1 19424.734,E2 19424.734} C_VEL
LIN {X 0,Y 434.299,Z 476.241,A -85,B 0,C 180,E1 19422.93,E2 19422.93} C_VEL
LIN {X 0,Y 437.114,Z 480.268,A -85,B 0,C 180,E1 19421.46,E2 19421.46} C_VEL
LIN {X 0,Y 439.61,Z 482.606,A -85,B 0,C 180,E1 19420.329,E2 19420.329} C_VEL
LIN {X 0,Y 446.992,Z 492.309,A -85,B 0,C 180,E1 19417.267,E2 19417.267} C_VEL
LIN {X 0,Y 452.308,Z 499.637,A -85,B 0,C 180,E1 19415.338,E2 19415.338} C_VEL
LIN {X 0,Y 458.323,Z 508.1,A -85,B 0,C 180,E1 19413.364,E2 19413.364} C_VEL
LIN {X 0,Y 466.579,Z 520.08,A -85,B 0,C 180,E1 19410.926,E2 19410.926} C_VEL
LIN {X 0,Y 476.653,Z 535.78,A -85,B 0,C 180,E1 19408.264,E2 19408.264} C_VEL
LIN {X 0,Y 486.066,Z 551.603,A -85,B 0,C 180,E1 19406.012,E2 19406.012} C_VEL
LIN {X 0,Y 492.825,Z 563.92,A -85,B 0,C 180,E1 19404.501,E2 19404.501} C_VEL
LIN {X 0,Y 480.875,Z 782.524,A -85,B 0,C 180,E1 19401.063,E2 19401.063} C_VEL
LIN {X 0,Y 477.713,Z 837.48,A -85,B 0,C 180,E1 19400.172,E2 19400.172} C_VEL
LIN {X 0,Y 474.955,Z 862.161,A -85,B 0,C 180,E1 19399.619,E2 19399.619} C_VEL
LIN {X 0,Y 471.608,Z 884.741,A -85,B 0,C 180,E1 19398.958,E2 19398.958} C_VEL
LIN {X 0,Y 467.204,Z 908.575,A -85,B 0,C 180,E1 19398.048,E2 19398.048} C_VEL
LIN {X 0,Y 462.833,Z 928.952,A -85,B 0,C 180,E1 19397.085,E2 19397.085} C_VEL
LIN {X 0,Y 456.949,Z 953.116,A -85,B 0,C 180,E1 19395.688,E2 19395.688} C_VEL
LIN {X 0,Y 451.713,Z 972.254,A -85,B 0,C 180,E1 19394.358,E2 19394.358} C_VEL
LIN {X 0,Y 445.63,Z 993.037,A -85,B 0,C 180,E1 19392.658,E2 19392.658} C_VEL
LIN {X 0,Y 439.639,Z 1011.807,A -85,B 0,C 180,E1 19390.835,E2 19390.835} C_VEL
LIN {X 0,Y 433.68,Z 1029.865,A -85,B 0,C 180,E1 19388.804,E2 19388.804} C_VEL
LIN {X 0,Y 427.464,Z 1047.791,A -85,B 0,C 180,E1 19386.422,E2 19386.422} C_VEL
LIN {X 0,Y 422,Z 1063.527,A -85,B 0,C 180,E1 19383.999,E2 19383.999} C_VEL
LIN {X 0,Y 416.684,Z 1078.89,A -85,B 0,C 180,E1 19381.22,E2 19381.22} C_VEL
LIN {X 0,Y 412.605,Z 1091.039,A -85,B 0,C 180,E1 19378.674,E2 19378.674} C_VEL
LIN {X 0,Y 408.356,Z 1104.526,A -85,B 0,C 180,E1 19375.373,E2 19375.373} C_VEL
LIN {X 0,Y 405.469,Z 1114.508,A -85,B 0,C 180,E1 19372.472,E2 19372.472} C_VEL
LIN {X 0,Y 403.05,Z 1124.342,A -85,B 0,C 180,E1 19369.115,E2 19369.115} C_VEL
LIN {X 0,Y 401.436,Z 1132.242,A -85,B 0,C 180,E1 19365.753,E2 19365.753} C_VEL
LIN {X 0,Y 400.53,Z 1138.385,A -85,B 0,C 180,E1 19362.544,E2 19362.544} C_VEL
LIN {X 0,Y 400.071,Z 1143.359,A -85,B 0,C 180,E1 19359.059,E2 19359.059} C_VEL
LIN {X 0,Y 399.981,Z 1146.247,A -85,B 0,C 180,E1 19356.171,E2 19356.171} C_VEL
LIN {X 0,Y 399.971,Z 1148.104,A -85,B 0,C 180,E1 19353.153,E2 19353.153} C_VEL
LIN {X 0,Y 400.001,Z 1148.694,A -85,B 0,C 180,E1 19349.857,E2 19349.857} C_VEL
LIN {X 0,Y 399.977,Z 1147.881,A -85,B 0,C 180,E1 19346.847,E2 19346.847} C_VEL
LIN {X 0,Y 399.983,Z 1146.106,A -85,B 0,C 180,E1 19344.117,E2 19344.117} C_VEL
LIN {X 0,Y 400.074,Z 1142.817,A -85,B 0,C 180,E1 19340.941,E2 19340.941} C_VEL
LIN {X 0,Y 400.487,Z 1137.73,A -85,B 0,C 180,E1 19337.601,E2 19337.601} C_VEL
LIN {X 0,Y 401.242,Z 1131.994,A -85,B 0,C 180,E1 19334.667,E2 19334.667} C_VEL
LIN {X 0,Y 402.708,Z 1123.974,A -85,B 0,C 180,E1 19331.319,E2 19331.319} C_VEL
LIN {X 0,Y 404.842,Z 1114.418,A -85,B 0,C 180,E1 19328.103,E2 19328.103} C_VEL
LIN {X 0,Y 407.812,Z 1103.242,A -85,B 0,C 180,E1 19324.902,E2 19324.902} C_VEL
LIN {X 0,Y 411.459,Z 1090.537,A -85,B 0,C 180,E1 19321.872,E2 19321.872} C_VEL
LIN {X 0,Y 415.527,Z 1077.434,A -85,B 0,C 180,E1 19319.166,E2 19319.166} C_VEL
LIN {X 0,Y 420.583,Z 1061.497,A -85,B 0,C 180,E1 19316.363,E2 19316.363} C_VEL
LIN {X 0,Y 425.402,Z 1046.566,A -85,B 0,C 180,E1 19314.095,E2 19314.095} C_VEL
LIN {X 0,Y 431.494,Z 1027.457,A -85,B 0,C 180,E1 19311.608,E2 19311.608} C_VEL
LIN {X 0,Y 436.76,Z 1010.339,A -85,B 0,C 180,E1 19309.704,E2 19309.704} C_VEL
LIN {X 0,Y 442.878,Z 989.499,A -85,B 0,C 180,E1 19307.716,E2 19307.716} C_VEL
LIN {X 0,Y 448.151,Z 970.062,A -85,B 0,C 180,E1 19306.15,E2 19306.15} C_VEL
LIN {X 0,Y 453.584,Z 948.696,A -85,B 0,C 180,E1 19304.685,E2 19304.685} C_VEL
LIN {X 0,Y 458.507,Z 926.47,A -85,B 0,C 180,E1 19303.432,E2 19303.432} C_VEL
LIN {X 0,Y 463.139,Z 903.131,A -85,B 0,C 180,E1 19302.345,E2 19302.345} C_VEL
LIN {X 0,Y 467.006,Z 879.356,A -85,B 0,C 180,E1 19301.486,E2 19301.486} C_VEL
LIN {X 0,Y 470.284,Z 854.938,A -85,B 0,C 180,E1 19300.802,E2 19300.802} C_VEL
LIN {X 0,Y 472.422,Z 830.38,A -85,B 0,C 180,E1 19300.305,E2 19300.305} C_VEL
LIN {X 0,Y 483.689,Z 607.043,A -85,B 0,C 180,E1 19296.776,E2 19296.776} C_VEL
LIN {X 0,Y 485.995,Z 559.651,A -85,B 0,C 180,E1 19296.009,E2 19296.009} C_VEL
LIN {X 0,Y 475.656,Z 540.973,A -85,B 0,C 180,E1 19293.889,E2 19293.889} C_VEL
LIN {X 0,Y 464.829,Z 522.995,A -85,B 0,C 180,E1 19291.479,E2 19291.479} C_VEL
LIN {X 0,Y 454.736,Z 507.381,A -85,B 0,C 180,E1 19289.002,E2 19289.002} C_VEL
LIN {X 0,Y 445.011,Z 493.286,A -85,B 0,C 180,E1 19286.344,E2 19286.344} C_VEL
LIN {X 0,Y 437.189,Z 482.599,A -85,B 0,C 180,E1 19283.951,E2 19283.951} C_VEL
LIN {X 0,Y 430.506,Z 473.972,A -85,B 0,C 180,E1 19281.672,E2 19281.672} C_VEL
LIN {X 0,Y 427.072,Z 470.2,A -85,B 0,C 180,E1 19280.417,E2 19280.417} C_VEL
LIN {X 0,Y 425.636,Z 468.149,A -85,B 0,C 180,E1 19279.844,E2 19279.844} C_VEL
LIN {X 0,Y 422.269,Z 464.927,A -85,B 0,C 180,E1 19278.5,E2 19278.5} C_VEL
LIN {X 0,Y 420.569,Z 462.077,A -85,B 0,C 180,E1 19277.717,E2 19277.717} C_VEL
LIN {X 0,Y 417.188,Z 459.522,A -85,B 0,C 180,E1 19276.214,E2 19276.214} C_VEL
LIN {X 0,Y 415.08,Z 455.893,A -85,B 0,C 180,E1 19275.08,E2 19275.08} C_VEL
LIN {X 0,Y 410.977,Z 452.878,A -85,B 0,C 180,E1 19272.863,E2 19272.863} C_VEL
LIN {X 0,Y 408.693,Z 449.066,A -85,B 0,C 180,E1 19271.287,E2 19271.287} C_VEL
LIN {X 0,Y 404.482,Z 446.189,A -85,B 0,C 180,E1 19268.1,E2 19268.1} C_VEL
LIN {X 0,Y 402.785,Z 442.773,A -85,B 0,C 180,E1 19265.842,E2 19265.842} C_VEL
LIN {X 0,Y 402.661,Z 442.058,A -85,B 0,C 180,E1 19263.702,E2 19263.702} C_VEL
LIN {X 0,Y 402.67,Z 442.053,A -85,B 0,C 180,E1 19259.715,E2 19259.715} C_VEL
LIN {X 0,Y 402.657,Z 442.039,A -85,B 0,C 180,E1 19255.728,E2 19255.728} C_VEL
LIN {X 0,Y 402.666,Z 442.133,A -85,B 0,C 180,E1 19251.863,E2 19251.863} C_VEL
LIN {X 0,Y 402.863,Z 443.207,A -85,B 0,C 180,E1 19250.283,E2 19250.283} C_VEL
LIN {X 0,Y 404.844,Z 446.64,A -85,B 0,C 180,E1 19248.026,E2 19248.026} C_VEL
LIN {X 0,Y 408.975,Z 449.382,A -85,B 0,C 180,E1 19244.98,E2 19244.98} C_VEL
LIN {X 0,Y 411.185,Z 453.147,A -85,B 0,C 180,E1 19243.47,E2 19243.47} C_VEL
LIN {X 0,Y 414.411,Z 455.417,A -85,B 0,C 180,E1 19241.72,E2 19241.72} C_VEL
LIN {X 0,Y 415.123,Z 456.066,A -85,B 0,C 180,E1 19241.352,E2 19241.352} C_VEL
LIN {X 0,Y 417.186,Z 459.511,A -85,B 0,C 180,E1 19240.248,E2 19240.248} C_VEL
LIN {X 0,Y 420.924,Z 462.669,A -85,B 0,C 180,E1 19238.578,E2 19238.578} C_VEL
LIN {X 0,Y 423.508,Z 466.45,A -85,B 0,C 180,E1 19237.439,E2 19237.439} C_VEL
LIN {X 0,Y 426.228,Z 468.826,A -85,B 0,C 180,E1 19236.386,E2 19236.386} C_VEL
LIN {X 0,Y 429.282,Z 472.967,A -85,B 0,C 180,E1 19235.212,E2 19235.212} C_VEL
LIN {X 0,Y 431.514,Z 475.156,A -85,B 0,C 180,E1 19234.432,E2 19234.432} C_VEL
LIN {X 0,Y 435.048,Z 479.531,A -85,B 0,C 180,E1 19233.226,E2 19233.226} C_VEL
LIN {X 0,Y 436.759,Z 481.594,A -85,B 0,C 180,E1 19232.669,E2 19232.669} C_VEL
LIN {X 0,Y 441.51,Z 487.453,A -85,B 0,C 180,E1 19231.196,E2 19231.196} C_VEL
LIN {X 0,Y 446.314,Z 493.487,A -85,B 0,C 180,E1 19229.804,E2 19229.804} C_VEL
LIN {X 0,Y 453.53,Z 502.791,A -85,B 0,C 180,E1 19227.867,E2 19227.867} C_VEL
LIN {X 0,Y 463.964,Z 517.015,A -85,B 0,C 180,E1 19225.323,E2 19225.323} C_VEL
LIN {X 0,Y 474.201,Z 531.84,A -85,B 0,C 180,E1 19223.062,E2 19223.062} C_VEL
LIN {X 0,Y 486.43,Z 551.052,A -85,B 0,C 180,E1 19220.595,E2 19220.595} C_VEL
LIN {X 0,Y 473.83,Z 797.809,A -85,B 0,C 180,E1 19216.725,E2 19216.725} C_VEL
LIN {X 0,Y 471.996,Z 823.586,A -85,B 0,C 180,E1 19216.241,E2 19216.241} C_VEL
LIN {X 0,Y 469.666,Z 845.401,A -85,B 0,C 180,E1 19215.685,E2 19215.685} C_VEL
LIN {X 0,Y 466.156,Z 870.25,A -85,B 0,C 180,E1 19214.843,E2 19214.843} C_VEL
LIN {X 0,Y 462.605,Z 890.798,A -85,B 0,C 180,E1 19213.965,E2 19213.965} C_VEL
LIN {X 0,Y 457.76,Z 914.812,A -85,B 0,C 180,E1 19212.706,E2 19212.706} C_VEL
LIN {X 0,Y 453.129,Z 934.6,A -85,B 0,C 180,E1 19211.452,E2 19211.452} C_VEL
LIN {X 0,Y 447.711,Z 955.823,A -85,B 0,C 180,E1 19209.864,E2 19209.864} C_VEL
LIN {X 0,Y 442.342,Z 974.68,A -85,B 0,C 180,E1 19208.187,E2 19208.187} C_VEL
LIN {X 0,Y 436.95,Z 992.661,A -85,B 0,C 180,E1 19206.341,E2 19206.341} C_VEL
LIN {X 0,Y 431.114,Z 1010.874,A -85,B 0,C 180,E1 19204.144,E2 19204.144} C_VEL
LIN {X 0,Y 426.108,Z 1026.032,A -85,B 0,C 180,E1 19202.028,E2 19202.028} C_VEL
LIN {X 0,Y 420.288,Z 1043.392,A -85,B 0,C 180,E1 19199.19,E2 19199.19} C_VEL
LIN {X 0,Y 415.945,Z 1056.333,A -85,B 0,C 180,E1 19196.714,E2 19196.714} C_VEL
LIN {X 0,Y 411.285,Z 1070.656,A -85,B 0,C 180,E1 19193.497,E2 19193.497} C_VEL
LIN {X 0,Y 407.975,Z 1081.297,A -85,B 0,C 180,E1 19190.666,E2 19190.666} C_VEL
LIN {X 0,Y 404.919,Z 1092.143,A -85,B 0,C 180,E1 19187.237,E2 19187.237} C_VEL
LIN {X 0,Y 402.968,Z 1099.974,A -85,B 0,C 180,E1 19184.22,E2 19184.22} C_VEL
LIN {X 0,Y 401.516,Z 1107.092,A -85,B 0,C 180,E1 19180.91,E2 19180.91} C_VEL
LIN {X 0,Y 400.639,Z 1112.47,A -85,B 0,C 180,E1 19177.601,E2 19177.601} C_VEL
LIN {X 0,Y 400.239,Z 1116.17,A -85,B 0,C 180,E1 19174.584,E2 19174.584} C_VEL
LIN {X 0,Y 400.035,Z 1118.968,A -85,B 0,C 180,E1 19171.121,E2 19171.121} C_VEL
LIN {X 0,Y 399.999,Z 1120.06,A -85,B 0,C 180,E1 19168.138,E2 19168.138} C_VEL
LIN {X 0,Y 399.996,Z 1120.094,A -85,B 0,C 180,E1 19165.412,E2 19165.412} C_VEL
LIN {X 0,Y 400.057,Z 1119.12,A -85,B 0,C 180,E1 19162.532,E2 19162.532} C_VEL
LIN {X 0,Y 400.305,Z 1116.46,A -85,B 0,C 180,E1 19159.007,E2 19159.007} C_VEL
LIN {X 0,Y 400.385,Z 1115.692,A -85,B 0,C 180,E1 19158.288,E2 19158.288} C_VEL
LIN {X 0,Y 399.552,Z 1114.593,A -85,B 0,C 180,E1 19157.195,E2 19157.195} C_VEL
LIN {X 0,Y 393.895,Z 1110.929,A -85,B 0,C 180,E1 19154.194,E2 19154.194} C_VEL
LIN {X 0,Y 393.521,Z 1109.53,A -85,B 0,C 180,E1 19153.325,E2 19153.325} C_VEL
LIN {X 0,Y 394.976,Z 1103.36,A -85,B 0,C 180,E1 19150.016,E2 19150.016} C_VEL
LIN {X 0,Y 397.253,Z 1095.168,A -85,B 0,C 180,E1 19146.566,E2 19146.566} C_VEL
LIN {X 0,Y 400.089,Z 1086.298,A -85,B 0,C 180,E1 19143.471,E2 19143.471} C_VEL
LIN {X 0,Y 404.262,Z 1074.385,A -85,B 0,C 180,E1 19140.025,E2 19140.025} C_VEL
LIN {X 0,Y 408.445,Z 1063.006,A -85,B 0,C 180,E1 19137.247,E2 19137.247} C_VEL
LIN {X 0,Y 414.247,Z 1047.704,A -85,B 0,C 180,E1 19134.088,E2 19134.088} C_VEL
LIN {X 0,Y 419.533,Z 1033.738,A -85,B 0,C 180,E1 19131.64,E2 19131.64} C_VEL
LIN {X 0,Y 426.283,Z 1015.68,A -85,B 0,C 180,E1 19128.946,E2 19128.946} C_VEL
LIN {X 0,Y 431.975,Z 999.838,A -85,B 0,C 180,E1 19126.934,E2 19126.934} C_VEL
LIN {X 0,Y 438.562,Z 980.676,A -85,B 0,C 180,E1 19124.841,E2 19124.841} C_VEL
LIN {X 0,Y 444.486,Z 961.959,A -85,B 0,C 180,E1 19123.115,E2 19123.115} C_VEL
LIN {X 0,Y 450.291,Z 942.282,A -85,B 0,C 180,E1 19121.554,E2 19121.554} C_VEL
LIN {X 0,Y 455.818,Z 921.175,A -85,B 0,C 180,E1 19120.16,E2 19120.16} C_VEL
LIN {X 0,Y 460.417,Z 901.605,A -85,B 0,C 180,E1 19119.069,E2 19119.069} C_VEL
LIN {X 0,Y 465.206,Z 877.833,A -85,B 0,C 180,E1 19117.975,E2 19117.975} C_VEL
LIN {X 0,Y 468.605,Z 857.394,A -85,B 0,C 180,E1 19117.222,E2 19117.222} C_VEL
LIN {X 0,Y 471.862,Z 833.495,A -85,B 0,C 180,E1 19116.527,E2 19116.527} C_VEL
LIN {X 0,Y 474.055,Z 809.349,A -85,B 0,C 180,E1 19116.023,E2 19116.023} C_VEL
LIN {X 0,Y 487.654,Z 571.425,A -85,B 0,C 180,E1 19112.264,E2 19112.264} C_VEL
LIN {X 0,Y 488.316,Z 559.238,A -85,B 0,C 180,E1 19112.063,E2 19112.063} C_VEL
LIN {X 0,Y 478.424,Z 543.887,A -85,B 0,C 180,E1 19109.795,E2 19109.795} C_VEL
LIN {X 0,Y 469.21,Z 530.58,A -85,B 0,C 180,E1 19107.475,E2 19107.475} C_VEL
LIN {X 0,Y 461.704,Z 520.283,A -85,B 0,C 180,E1 19105.392,E2 19105.392} C_VEL
LIN {X 0,Y 454.796,Z 511.219,A -85,B 0,C 180,E1 19103.278,E2 19103.278} C_VEL
LIN {X 0,Y 450.105,Z 505.309,A -85,B 0,C 180,E1 19101.708,E2 19101.708} C_VEL
LIN {X 0,Y 446.28,Z 500.483,A -85,B 0,C 180,E1 19100.321,E2 19100.321} C_VEL
LIN {X 0,Y 441.773,Z 494.94,A -85,B 0,C 180,E1 19098.542,E2 19098.542} C_VEL
LIN {X 0,Y 438.19,Z 490.59,A -85,B 0,C 180,E1 19096.983,E2 19096.983} C_VEL
LIN {X 0,Y 437.102,Z 489.29,A -85,B 0,C 180,E1 19096.479,E2 19096.479} C_VEL
LIN {X 0,Y 433.741,Z 485.578,A -85,B 0,C 180,E1 19094.826,E2 19094.826} C_VEL
LIN {X 0,Y 432.365,Z 483.431,A -85,B 0,C 180,E1 19094.053,E2 19094.053} C_VEL
LIN {X 0,Y 429.088,Z 480.6,A -85,B 0,C 180,E1 19092.175,E2 19092.175} C_VEL
LIN {X 0,Y 427.166,Z 477.234,A -85,B 0,C 180,E1 19090.793,E2 19090.793} C_VEL
LIN {X 0,Y 423.728,Z 474.73,A -85,B 0,C 180,E1 19088.14,E2 19088.14} C_VEL
LIN {X 0,Y 421.622,Z 470.87,A -85,B 0,C 180,E1 19085.716,E2 19085.716} C_VEL
LIN {X 0,Y 418.718,Z 469.315,A -85,B 0,C 180,E1 19079.59,E2 19079.59} C_VEL
LIN {X 0,Y 419.526,Z 469.853,A -85,B 0,C 180,E1 19074.941,E2 19074.941} C_VEL
LIN {X 0,Y 421.783,Z 471.042,A -85,B 0,C 180,E1 19071.548,E2 19071.548} C_VEL
LIN {X 0,Y 423.801,Z 474.791,A -85,B 0,C 180,E1 19069.258,E2 19069.258} C_VEL
LIN {X 0,Y 427.437,Z 477.628,A -85,B 0,C 180,E1 19066.472,E2 19066.472} C_VEL
LIN {X 0,Y 429.826,Z 481.414,A -85,B 0,C 180,E1 19064.829,E2 19064.829} C_VEL
LIN {X 0,Y 432.838,Z 484.051,A -85,B 0,C 180,E1 19063.147,E2 19063.147} C_VEL
LIN {X 0,Y 435.889,Z 488.225,A -85,B 0,C 180,E1 19061.545,E2 19061.545} C_VEL
LIN {X 0,Y 437.943,Z 490.204,A -85,B 0,C 180,E1 19060.598,E2 19060.598} C_VEL
LIN {X 0,Y 444.902,Z 499.458,A -85,B 0,C 180,E1 19057.643,E2 19057.643} C_VEL
LIN {X 0,Y 450.719,Z 507.618,A -85,B 0,C 180,E1 19055.49,E2 19055.49} C_VEL
LIN {X 0,Y 456.219,Z 515.534,A -85,B 0,C 180,E1 19053.652,E2 19053.652} C_VEL
LIN {X 0,Y 464.142,Z 527.26,A -85,B 0,C 180,E1 19051.263,E2 19051.263} C_VEL
LIN {X 0,Y 473.579,Z 542.182,A -85,B 0,C 180,E1 19048.708,E2 19048.708} C_VEL
LIN {X 0,Y 482.734,Z 557.817,A -85,B 0,C 180,E1 19046.46,E2 19046.46} C_VEL
LIN {X 0,Y 488.114,Z 567.77,A -85,B 0,C 180,E1 19045.218,E2 19045.218} C_VEL
LIN {X 0,Y 475.75,Z 787.039,A -85,B 0,C 180,E1 19041.754,E2 19041.754} C_VEL
LIN {X 0,Y 472.705,Z 837.83,A -85,B 0,C 180,E1 19040.923,E2 19040.923} C_VEL
LIN {X 0,Y 469.858,Z 862.353,A -85,B 0,C 180,E1 19040.369,E2 19040.369} C_VEL
LIN {X 0,Y 466.282,Z 885.799,A -85,B 0,C 180,E1 19039.677,E2 19039.677} C_VEL
LIN {X 0,Y 461.869,Z 908.759,A -85,B 0,C 180,E1 19038.79,E2 19038.79} C_VEL
LIN {X 0,Y 457.383,Z 929.08,A -85,B 0,C 180,E1 19037.825,E2 19037.825} C_VEL
LIN {X 0,Y 451.328,Z 953.159,A -85,B 0,C 180,E1 19036.423,E2 19036.423} C_VEL
LIN {X 0,Y 445.761,Z 972.879,A -85,B 0,C 180,E1 19035.042,E2 19035.042} C_VEL
LIN {X 0,Y 439.118,Z 994.633,A -85,B 0,C 180,E1 19033.226,E2 19033.226} C_VEL
LIN {X 0,Y 433.266,Z 1012.346,A -85,B 0,C 180,E1 19031.479,E2 19031.479} C_VEL
LIN {X 0,Y 426.817,Z 1031.164,A -85,B 0,C 180,E1 19029.323,E2 19029.323} C_VEL
LIN {X 0,Y 420.574,Z 1048.435,A -85,B 0,C 180,E1 19026.977,E2 19026.977} C_VEL
LIN {X 0,Y 414.579,Z 1065.073,A -85,B 0,C 180,E1 19024.358,E2 19024.358} C_VEL
LIN {X 0,Y 409.108,Z 1080.135,A -85,B 0,C 180,E1 19021.536,E2 19021.536} C_VEL
LIN {X 0,Y 404.294,Z 1094.061,A -85,B 0,C 180,E1 19018.511,E2 19018.511} C_VEL
LIN {X 0,Y 400.212,Z 1106.412,A -85,B 0,C 180,E1 19015.292,E2 19015.292} C_VEL
LIN {X 0,Y 397.091,Z 1117.092,A -85,B 0,C 180,E1 19012.036,E2 19012.036} C_VEL
LIN {X 0,Y 394.742,Z 1126.273,A -85,B 0,C 180,E1 19008.612,E2 19008.612} C_VEL
LIN {X 0,Y 393.328,Z 1133.242,A -85,B 0,C 180,E1 19005.481,E2 19005.481} C_VEL
LIN {X 0,Y 392.378,Z 1139.737,A -85,B 0,C 180,E1 19001.763,E2 19001.763} C_VEL
LIN {X 0,Y 392.061,Z 1143.592,A -85,B 0,C 180,E1 18998.802,E2 18998.802} C_VEL
LIN {X 0,Y 391.967,Z 1146.449,A -85,B 0,C 180,E1 18995.71,E2 18995.71} C_VEL
LIN {X 0,Y 391.987,Z 1148.133,A -85,B 0,C 180,E1 18992.339,E2 18992.339} C_VEL
LIN {X 0,Y 391.996,Z 1148.315,A -85,B 0,C 180,E1 18989.269,E2 18989.269} C_VEL
LIN {X 0,Y 391.989,Z 1147.445,A -85,B 0,C 180,E1 18986.49,E2 18986.49} C_VEL
LIN {X 0,Y 391.994,Z 1145.332,A -85,B 0,C 180,E1 18983.409,E2 18983.409} C_VEL
LIN {X 0,Y 392.169,Z 1141.287,A -85,B 0,C 180,E1 18979.867,E2 18979.867} C_VEL
LIN {X 0,Y 392.664,Z 1136.35,A -85,B 0,C 180,E1 18976.751,E2 18976.751} C_VEL
LIN {X 0,Y 393.747,Z 1129.472,A -85,B 0,C 180,E1 18973.324,E2 18973.324} C_VEL
LIN {X 0,Y 395.447,Z 1121.115,A -85,B 0,C 180,E1 18970.041,E2 18970.041} C_VEL
LIN {X 0,Y 397.933,Z 1111.218,A -85,B 0,C 180,E1 18966.765,E2 18966.765} C_VEL
LIN {X 0,Y 401.295,Z 1099.343,A -85,B 0,C 180,E1 18963.512,E2 18963.512} C_VEL
LIN {X 0,Y 404.974,Z 1087.526,A -85,B 0,C 180,E1 18960.734,E2 18960.734} C_VEL
LIN {X 0,Y 409.892,Z 1072.434,A -85,B 0,C 180,E1 18957.708,E2 18957.708} C_VEL
LIN {X 0,Y 414.557,Z 1058.46,A -85,B 0,C 180,E1 18955.304,E2 18955.304} C_VEL
LIN {X 0,Y 420.511,Z 1040.724,A -85,B 0,C 180,E1 18952.675,E2 18952.675} C_VEL
LIN {X 0,Y 425.983,Z 1023.944,A -85,B 0,C 180,E1 18950.556,E2 18950.556} C_VEL
LIN {X 0,Y 432.048,Z 1004.888,A -85,B 0,C 180,E1 18948.476,E2 18948.476} C_VEL
LIN {X 0,Y 437.918,Z 985.031,A -85,B 0,C 180,E1 18946.655,E2 18946.655} C_VEL
LIN {X 0,Y 443.583,Z 964.716,A -85,B 0,C 180,E1 18945.056,E2 18945.056} C_VEL
LIN {X 0,Y 449.038,Z 942.981,A -85,B 0,C 180,E1 18943.64,E2 18943.64} C_VEL
LIN {X 0,Y 453.714,Z 922.213,A -85,B 0,C 180,E1 18942.5,E2 18942.5} C_VEL
LIN {X 0,Y 458.426,Z 898.079,A -85,B 0,C 180,E1 18941.43,E2 18941.43} C_VEL
LIN {X 0,Y 461.978,Z 876.469,A -85,B 0,C 180,E1 18940.67,E2 18940.67} C_VEL
LIN {X 0,Y 465.426,Z 849.763,A -85,B 0,C 180,E1 18939.961,E2 18939.961} C_VEL
LIN {X 0,Y 467.304,Z 827.403,A -85,B 0,C 180,E1 18939.52,E2 18939.52} C_VEL
LIN {X 0,Y 478.947,Z 603.304,A -85,B 0,C 180,E1 18935.964,E2 18935.964} C_VEL
LIN {X 0,Y 480.942,Z 563.245,A -85,B 0,C 180,E1 18935.308,E2 18935.308} C_VEL
LIN {X 0,Y 470.741,Z 544.72,A -85,B 0,C 180,E1 18933.14,E2 18933.14} C_VEL
LIN {X 0,Y 459.98,Z 526.737,A -85,B 0,C 180,E1 18930.647,E2 18930.647} C_VEL
LIN {X 0,Y 450.561,Z 512.242,A -85,B 0,C 180,E1 18928.245,E2 18928.245} C_VEL
LIN {X 0,Y 442.29,Z 500.028,A -85,B 0,C 180,E1 18925.905,E2 18925.905} C_VEL
LIN {X 0,Y 434.607,Z 489.389,A -85,B 0,C 180,E1 18923.49,E2 18923.49} C_VEL
LIN {X 0,Y 428.478,Z 481.364,A -85,B 0,C 180,E1 18921.349,E2 18921.349} C_VEL
LIN {X 0,Y 424.866,Z 477.203,A -85,B 0,C 180,E1 18919.989,E2 18919.989} C_VEL
LIN {X 0,Y 423.68,Z 475.607,A -85,B 0,C 180,E1 18919.508,E2 18919.508} C_VEL
LIN {X 0,Y 420.24,Z 472.068,A -85,B 0,C 180,E1 18918.09,E2 18918.09} C_VEL
LIN {X 0,Y 418.695,Z 469.635,A -85,B 0,C 180,E1 18917.368,E2 18917.368} C_VEL
LIN {X 0,Y 415.271,Z 466.73,A -85,B 0,C 180,E1 18915.788,E2 18915.788} C_VEL
LIN {X 0,Y 413.335,Z 463.364,A -85,B 0,C 180,E1 18914.715,E2 18914.715} C_VEL
LIN {X 0,Y 409.776,Z 460.813,A -85,B 0,C 180,E1 18912.758,E2 18912.758} C_VEL
LIN {X 0,Y 407.797,Z 457.443,A -85,B 0,C 180,E1 18911.384,E2 18911.384} C_VEL
LIN {X 0,Y 406.697,Z 456.507,A -85,B 0,C 180,E1 18910.626,E2 18910.626} C_VEL
LIN {X 0,Y 403.208,Z 453.894,A -85,B 0,C 180,E1 18907.839,E2 18907.839} C_VEL
LIN {X 0,Y 401.164,Z 450.348,A -85,B 0,C 180,E1 18905.435,E2 18905.435} C_VEL
LIN {X 0,Y 398.642,Z 448.978,A -85,B 0,C 180,E1 18901.006,E2 18901.006} C_VEL
LIN {X 0,Y 398.497,Z 448.873,A -85,B 0,C 180,E1 18895.971,E2 18895.971} C_VEL
LIN {X 0,Y 401.096,Z 450.305,A -85,B 0,C 180,E1 18891.109,E2 18891.109} C_VEL
LIN {X 0,Y 402.268,Z 452.464,A -85,B 0,C 180,E1 18889.618,E2 18889.618} C_VEL
LIN {X 0,Y 404.539,Z 455.226,A -85,B 0,C 180,E1 18887.437,E2 18887.437} C_VEL
LIN {X 0,Y 407.607,Z 457.089,A -85,B 0,C 180,E1 18885.219,E2 18885.219} C_VEL
LIN {X 0,Y 409.556,Z 460.582,A -85,B 0,C 180,E1 18883.84,E2 18883.84} C_VEL
LIN {X 0,Y 412.679,Z 463.048,A -85,B 0,C 180,E1 18882.079,E2 18882.079} C_VEL
LIN {X 0,Y 413.509,Z 463.757,A -85,B 0,C 180,E1 18881.642,E2 18881.642} C_VEL
LIN {X 0,Y 415.818,Z 467.366,A -85,B 0,C 180,E1 18880.4,E2 18880.4} C_VEL
LIN {X 0,Y 419.142,Z 470.24,A -85,B 0,C 180,E1 18878.886,E2 18878.886} C_VEL
LIN {X 0,Y 421.928,Z 474.162,A -85,B 0,C 180,E1 18877.644,E2 18877.644} C_VEL
LIN {X 0,Y 424.36,Z 476.408,A -85,B 0,C 180,E1 18876.681,E2 18876.681} C_VEL
LIN {X 0,Y 427.644,Z 480.691,A -85,B 0,C 180,E1 18875.406,E2 18875.406} C_VEL
LIN {X 0,Y 429.489,Z 482.596,A -85,B 0,C 180,E1 18874.746,E2 18874.746} C_VEL
LIN {X 0,Y 433.36,Z 487.258,A -85,B 0,C 180,E1 18873.409,E2 18873.409} C_VEL
LIN {X 0,Y 439.452,Z 495.032,A -85,B 0,C 180,E1 18871.457,E2 18871.457} C_VEL
LIN {X 0,Y 444.208,Z 501.071,A -85,B 0,C 180,E1 18870.056,E2 18870.056} C_VEL
LIN {X 0,Y 450.915,Z 509.854,A -85,B 0,C 180,E1 18868.22,E2 18868.22} C_VEL
LIN {X 0,Y 460.99,Z 523.776,A -85,B 0,C 180,E1 18865.709,E2 18865.709} C_VEL
LIN {X 0,Y 470.983,Z 538.433,A -85,B 0,C 180,E1 18863.452,E2 18863.452} C_VEL
LIN {X 0,Y 481.378,Z 555.085,A -85,B 0,C 180,E1 18861.289,E2 18861.289} C_VEL
LIN {X 0,Y 468.121,Z 805.312,A -85,B 0,C 180,E1 18857.333,E2 18857.333} C_VEL
LIN {X 0,Y 466.38,Z 827.022,A -85,B 0,C 180,E1 18856.899,E2 18856.899} C_VEL
LIN {X 0,Y 463.541,Z 851.592,A -85,B 0,C 180,E1 18856.233,E2 18856.233} C_VEL
LIN {X 0,Y 460.365,Z 872.416,A -85,B 0,C 180,E1 18855.492,E2 18855.492} C_VEL
LIN {X 0,Y 456.602,Z 893.419,A -85,B 0,C 180,E1 18854.576,E2 18854.576} C_VEL
LIN {X 0,Y 451.701,Z 916.565,A -85,B 0,C 180,E1 18853.332,E2 18853.332} C_VEL
LIN {X 0,Y 447.171,Z 935.317,A -85,B 0,C 180,E1 18852.13,E2 18852.13} C_VEL
LIN {X 0,Y 441.377,Z 957.187,A -85,B 0,C 180,E1 18850.469,E2 18850.469} C_VEL
LIN {X 0,Y 435.858,Z 975.946,A -85,B 0,C 180,E1 18848.777,E2 18848.777} C_VEL
LIN {X 0,Y 429.959,Z 994.961,A -85,B 0,C 180,E1 18846.786,E2 18846.786} C_VEL
LIN {X 0,Y 423.949,Z 1012.899,A -85,B 0,C 180,E1 18844.557,E2 18844.557} C_VEL
LIN {X 0,Y 418.066,Z 1030.146,A -85,B 0,C 180,E1 18842.07,E2 18842.07} C_VEL
LIN {X 0,Y 412.702,Z 1045.377,A -85,B 0,C 180,E1 18839.461,E2 18839.461} C_VEL
LIN {X 0,Y 407.809,Z 1059.534,A -85,B 0,C 180,E1 18836.66,E2 18836.66} C_VEL
LIN {X 0,Y 403.48,Z 1072.207,A -85,B 0,C 180,E1 18833.67,E2 18833.67} C_VEL
LIN {X 0,Y 399.946,Z 1083.22,A -85,B 0,C 180,E1 18830.641,E2 18830.641} C_VEL
LIN {X 0,Y 396.965,Z 1093.321,A -85,B 0,C 180,E1 18827.291,E2 18827.291} C_VEL
LIN {X 0,Y 395.061,Z 1100.695,A -85,B 0,C 180,E1 18824.361,E2 18824.361} C_VEL
LIN {X 0,Y 393.503,Z 1107.945,A -85,B 0,C 180,E1 18820.838,E2 18820.838} C_VEL
LIN {X 0,Y 392.654,Z 1113.009,A -85,B 0,C 180,E1 18817.609,E2 18817.609} C_VEL
LIN {X 0,Y 392.229,Z 1116.805,A -85,B 0,C 180,E1 18814.386,E2 18814.386} C_VEL
LIN {X 0,Y 392.036,Z 1119.39,A -85,B 0,C 180,E1 18810.877,E2 18810.877} C_VEL
LIN {X 0,Y 392.005,Z 1120.373,A -85,B 0,C 180,E1 18807.954,E2 18807.954} C_VEL
LIN {X 0,Y 392.005,Z 1120.331,A -85,B 0,C 180,E1 18805.025,E2 18805.025} C_VEL
LIN {X 0,Y 392.129,Z 1119.011,A -85,B 0,C 180,E1 18801.637,E2 18801.637} C_VEL
LIN {X 0,Y 392.385,Z 1116.294,A -85,B 0,C 180,E1 18798.386,E2 18798.386} C_VEL
LIN {X 0,Y 392.919,Z 1112.714,A -85,B 0,C 180,E1 18795.408,E2 18795.408} C_VEL
LIN {X 0,Y 393.521,Z 1109.53,A -85,B 0,C 180,E1 18793.325,E2 18793.325} C_VEL
LIN {X 0,Y 392.922,Z 1107.822,A -85,B 0,C 180,E1 18792.227,E2 18792.227} C_VEL
LIN {X 0,Y 388.094,Z 1102.649,A -85,B 0,C 180,E1 18789.196,E2 18789.196} C_VEL
LIN {X 0,Y 388.002,Z 1100.782,A -85,B 0,C 180,E1 18788.333,E2 18788.333} C_VEL
LIN {X 0,Y 390.45,Z 1092.963,A -85,B 0,C 180,E1 18785.166,E2 18785.166} C_VEL
LIN {X 0,Y 394.106,Z 1082.466,A -85,B 0,C 180,E1 18781.677,E2 18781.677} C_VEL
LIN {X 0,Y 397.922,Z 1072.262,A -85,B 0,C 180,E1 18778.826,E2 18778.826} C_VEL
LIN {X 0,Y 403.287,Z 1058.55,A -85,B 0,C 180,E1 18775.577,E2 18775.577} C_VEL
LIN {X 0,Y 408.502,Z 1045.324,A -85,B 0,C 180,E1 18772.935,E2 18772.935} C_VEL
LIN {X 0,Y 414.648,Z 1029.891,A -85,B 0,C 180,E1 18770.281,E2 18770.281} C_VEL
LIN {X 0,Y 420.83,Z 1013.695,A -85,B 0,C 180,E1 18767.93,E2 18767.93} C_VEL
LIN {X 0,Y 427.009,Z 997.081,A -85,B 0,C 180,E1 18765.842,E2 18765.842} C_VEL
LIN {X 0,Y 433.658,Z 977.965,A -85,B 0,C 180,E1 18763.806,E2 18763.806} C_VEL
LIN {X 0,Y 439.399,Z 960.342,A -85,B 0,C 180,E1 18762.199,E2 18762.199} C_VEL
LIN {X 0,Y 445.862,Z 938.617,A -85,B 0,C 180,E1 18760.514,E2 18760.514} C_VEL
LIN {X 0,Y 451.156,Z 918.738,A -85,B 0,C 180,E1 18759.232,E2 18759.232} C_VEL
LIN {X 0,Y 456.407,Z 896.611,A -85,B 0,C 180,E1 18758.029,E2 18758.029} C_VEL
LIN {X 0,Y 460.773,Z 874.427,A -85,B 0,C 180,E1 18757.058,E2 18757.058} C_VEL
LIN {X 0,Y 464.252,Z 853.663,A -85,B 0,C 180,E1 18756.32,E2 18756.32} C_VEL
LIN {X 0,Y 467.509,Z 828.283,A -85,B 0,C 180,E1 18755.63,E2 18755.63} C_VEL
LIN {X 0,Y 469.431,Z 806.546,A -85,B 0,C 180,E1 18755.195,E2 18755.195} C_VEL
LIN {X 0,Y 483.725,Z 563.572,A -85,B 0,C 180,E1 18751.349,E2 18751.349} C_VEL
LIN {X 0,Y 475.072,Z 549.958,A -85,B 0,C 180,E1 18749.298,E2 18749.298} C_VEL
LIN {X 0,Y 466.332,Z 537.167,A -85,B 0,C 180,E1 18747.037,E2 18747.037} C_VEL
LIN {X 0,Y 459.053,Z 527.03,A -85,B 0,C 180,E1 18744.962,E2 18744.962} C_VEL
LIN {X 0,Y 452.175,Z 517.943,A -85,B 0,C 180,E1 18742.801,E2 18742.801} C_VEL
LIN {X 0,Y 447.926,Z 512.468,A -85,B 0,C 180,E1 18741.338,E2 18741.338} C_VEL
LIN {X 0,Y 444.328,Z 507.857,A -85,B 0,C 180,E1 18740.002,E2 18740.002} C_VEL
LIN {X 0,Y 439.897,Z 502.347,A -85,B 0,C 180,E1 18738.212,E2 18738.212} C_VEL
LIN {X 0,Y 436.262,Z 497.726,A -85,B 0,C 180,E1 18736.58,E2 18736.58} C_VEL
LIN {X 0,Y 432.155,Z 493.117,A -85,B 0,C 180,E1 18734.539,E2 18734.539} C_VEL
LIN {X 0,Y 430.916,Z 491.165,A -85,B 0,C 180,E1 18733.828,E2 18733.828} C_VEL
LIN {X 0,Y 427.604,Z 488.146,A -85,B 0,C 180,E1 18731.875,E2 18731.875} C_VEL
LIN {X 0,Y 425.811,Z 485.018,A -85,B 0,C 180,E1 18730.554,E2 18730.554} C_VEL
LIN {X 0,Y 422.467,Z 482.433,A -85,B 0,C 180,E1 18727.89,E2 18727.89} C_VEL
LIN {X 0,Y 420.427,Z 478.679,A -85,B 0,C 180,E1 18725.459,E2 18725.459} C_VEL
LIN {X 0,Y 417.72,Z 477.235,A -85,B 0,C 180,E1 18719.314,E2 18719.314} C_VEL
LIN {X 0,Y 418.823,Z 477.93,A -85,B 0,C 180,E1 18714.383,E2 18714.383} C_VEL
LIN {X 0,Y 420.699,Z 478.934,A -85,B 0,C 180,E1 18711.664,E2 18711.664} C_VEL
LIN {X 0,Y 422.543,Z 482.511,A -85,B 0,C 180,E1 18709.501,E2 18709.501} C_VEL
LIN {X 0,Y 426.089,Z 485.377,A -85,B 0,C 180,E1 18706.704,E2 18706.704} C_VEL
LIN {X 0,Y 428.54,Z 489.224,A -85,B 0,C 180,E1 18704.99,E2 18704.99} C_VEL
LIN {X 0,Y 431.332,Z 491.734,A -85,B 0,C 180,E1 18703.399,E2 18703.399} C_VEL
LIN {X 0,Y 434.403,Z 495.918,A -85,B 0,C 180,E1 18701.757,E2 18701.757} C_VEL
LIN {X 0,Y 436.353,Z 497.897,A -85,B 0,C 180,E1 18700.837,E2 18700.837} C_VEL
LIN {X 0,Y 442.905,Z 506.732,A -85,B 0,C 180,E1 18697.991,E2 18697.991} C_VEL
LIN {X 0,Y 449.912,Z 516.614,A -85,B 0,C 180,E1 18695.373,E2 18695.373} C_VEL
LIN {X 0,Y 459.363,Z 530.682,A -85,B 0,C 180,E1 18692.308,E2 18692.308} C_VEL
LIN {X 0,Y 469.278,Z 546.476,A -85,B 0,C 180,E1 18689.493,E2 18689.493} C_VEL
LIN {X 0,Y 479.046,Z 563.295,A -85,B 0,C 180,E1 18687.008,E2 18687.008} C_VEL
LIN {X 0,Y 483.476,Z 571.686,A -85,B 0,C 180,E1 18685.948,E2 18685.948} C_VEL
LIN {X 0,Y 470.786,Z 789.901,A -85,B 0,C 180,E1 18682.486,E2 18682.486} C_VEL
LIN {X 0,Y 467.796,Z 837.909,A -85,B 0,C 180,E1 18681.695,E2 18681.695} C_VEL
LIN {X 0,Y 464.858,Z 862.455,A -85,B 0,C 180,E1 18681.137,E2 18681.137} C_VEL
LIN {X 0,Y 461.124,Z 886.277,A -85,B 0,C 180,E1 18680.431,E2 18680.431} C_VEL
LIN {X 0,Y 456.614,Z 908.951,A -85,B 0,C 180,E1 18679.549,E2 18679.549} C_VEL
LIN {X 0,Y 451.75,Z 930.34,A -85,B 0,C 180,E1 18678.524,E2 18678.524} C_VEL
LIN {X 0,Y 445.785,Z 953.202,A -85,B 0,C 180,E1 18677.177,E2 18677.177} C_VEL
LIN {X 0,Y 440.312,Z 972.024,A -85,B 0,C 180,E1 18675.857,E2 18675.857} C_VEL
LIN {X 0,Y 433.582,Z 993.469,A -85,B 0,C 180,E1 18674.071,E2 18674.071} C_VEL
LIN {X 0,Y 427.369,Z 1011.671,A -85,B 0,C 180,E1 18672.272,E2 18672.272} C_VEL
LIN {X 0,Y 420.681,Z 1030.548,A -85,B 0,C 180,E1 18670.1,E2 18670.1} C_VEL
LIN {X 0,Y 414.369,Z 1047.38,A -85,B 0,C 180,E1 18667.801,E2 18667.801} C_VEL
LIN {X 0,Y 408.708,Z 1062.396,A -85,B 0,C 180,E1 18665.438,E2 18665.438} C_VEL
LIN {X 0,Y 402.597,Z 1078.554,A -85,B 0,C 180,E1 18662.443,E2 18662.443} C_VEL
LIN {X 0,Y 397.907,Z 1091.318,A -85,B 0,C 180,E1 18659.672,E2 18659.672} C_VEL
LIN {X 0,Y 393.257,Z 1104.642,A -85,B 0,C 180,E1 18656.258,E2 18656.258} C_VEL
LIN {X 0,Y 390.092,Z 1114.547,A -85,B 0,C 180,E1 18653.25,E2 18653.25} C_VEL
LIN {X 0,Y 387.317,Z 1124.599,A -85,B 0,C 180,E1 18649.609,E2 18649.609} C_VEL
LIN {X 0,Y 385.683,Z 1131.762,A -85,B 0,C 180,E1 18646.415,E2 18646.415} C_VEL
LIN {X 0,Y 384.606,Z 1138.152,A -85,B 0,C 180,E1 18642.92,E2 18642.92} C_VEL
LIN {X 0,Y 384.095,Z 1142.902,A -85,B 0,C 180,E1 18639.379,E2 18639.379} C_VEL
LIN {X 0,Y 383.984,Z 1145.829,A -85,B 0,C 180,E1 18636.279,E2 18636.279} C_VEL
LIN {X 0,Y 383.977,Z 1147.764,A -85,B 0,C 180,E1 18632.836,E2 18632.836} C_VEL
LIN {X 0,Y 384.001,Z 1148.072,A -85,B 0,C 180,E1 18629.552,E2 18629.552} C_VEL
LIN {X 0,Y 383.988,Z 1147.288,A -85,B 0,C 180,E1 18626.716,E2 18626.716} C_VEL
LIN {X 0,Y 383.994,Z 1145.496,A -85,B 0,C 180,E1 18623.871,E2 18623.871} C_VEL
LIN {X 0,Y 384.119,Z 1142.018,A -85,B 0,C 180,E1 18620.41,E2 18620.41} C_VEL
LIN {X 0,Y 384.621,Z 1136.802,A -85,B 0,C 180,E1 18616.928,E2 18616.928} C_VEL
LIN {X 0,Y 385.569,Z 1130.718,A -85,B 0,C 180,E1 18613.735,E2 18613.735} C_VEL
LIN {X 0,Y 387.497,Z 1121.583,A -85,B 0,C 180,E1 18609.928,E2 18609.928} C_VEL
LIN {X 0,Y 389.771,Z 1112.725,A -85,B 0,C 180,E1 18606.89,E2 18606.89} C_VEL
LIN {X 0,Y 393.33,Z 1100.707,A -85,B 0,C 180,E1 18603.422,E2 18603.422} C_VEL
LIN {X 0,Y 397.071,Z 1089.066,A -85,B 0,C 180,E1 18600.591,E2 18600.591} C_VEL
LIN {X 0,Y 401.832,Z 1075.142,A -85,B 0,C 180,E1 18597.657,E2 18597.657} C_VEL
LIN {X 0,Y 407.136,Z 1059.733,A -85,B 0,C 180,E1 18594.922,E2 18594.922} C_VEL
LIN {X 0,Y 412.916,Z 1043.275,A -85,B 0,C 180,E1 18592.394,E2 18592.394} C_VEL
LIN {X 0,Y 418.988,Z 1025.326,A -85,B 0,C 180,E1 18590.062,E2 18590.062} C_VEL
LIN {X 0,Y 424.677,Z 1008.063,A -85,B 0,C 180,E1 18588.126,E2 18588.126} C_VEL
LIN {X 0,Y 431.251,Z 986.874,A -85,B 0,C 180,E1 18586.111,E2 18586.111} C_VEL
LIN {X 0,Y 436.677,Z 968.051,A -85,B 0,C 180,E1 18584.592,E2 18584.592} C_VEL
LIN {X 0,Y 442.939,Z 944.353,A -85,B 0,C 180,E1 18582.996,E2 18582.996} C_VEL
LIN {X 0,Y 447.698,Z 923.902,A -85,B 0,C 180,E1 18581.854,E2 18581.854} C_VEL
LIN {X 0,Y 452.684,Z 899.484,A -85,B 0,C 180,E1 18580.745,E2 18580.745} C_VEL
LIN {X 0,Y 456.438,Z 877.4,A -85,B 0,C 180,E1 18579.957,E2 18579.957} C_VEL
LIN {X 0,Y 459.864,Z 852.414,A -85,B 0,C 180,E1 18579.273,E2 18579.273} C_VEL
LIN {X 0,Y 461.953,Z 829.081,A -85,B 0,C 180,E1 18578.802,E2 18578.802} C_VEL
LIN {X 0,Y 473.948,Z 606.043,A -85,B 0,C 180,E1 18575.239,E2 18575.239} C_VEL
LIN {X 0,Y 476.025,Z 566.948,A -85,B 0,C 180,E1 18574.606,E2 18574.606} C_VEL
LIN {X 0,Y 465.729,Z 548.157,A -85,B 0,C 180,E1 18572.334,E2 18572.334} C_VEL
LIN {X 0,Y 456.105,Z 532.093,A -85,B 0,C 180,E1 18570.025,E2 18570.025} C_VEL
LIN {X 0,Y 447.625,Z 518.795,A -85,B 0,C 180,E1 18567.794,E2 18567.794} C_VEL
LIN {X 0,Y 439.695,Z 506.898,A -85,B 0,C 180,E1 18565.491,E2 18565.491} C_VEL
LIN {X 0,Y 432.054,Z 496.172,A -85,B 0,C 180,E1 18563.024,E2 18563.024} C_VEL
LIN {X 0,Y 426.466,Z 488.75,A -85,B 0,C 180,E1 18561.022,E2 18561.022} C_VEL
LIN {X 0,Y 422.76,Z 484.331,A -85,B 0,C 180,E1 18559.588,E2 18559.588} C_VEL
LIN {X 0,Y 421.415,Z 482.791,A -85,B 0,C 180,E1 18559.041,E2 18559.041} C_VEL
LIN {X 0,Y 418.022,Z 478.879,A -85,B 0,C 180,E1 18557.577,E2 18557.577} C_VEL
LIN {X 0,Y 416.84,Z 477.166,A -85,B 0,C 180,E1 18557.017,E2 18557.017} C_VEL
LIN {X 0,Y 413.507,Z 474.092,A -85,B 0,C 180,E1 18555.426,E2 18555.426} C_VEL
LIN {X 0,Y 411.591,Z 470.978,A -85,B 0,C 180,E1 18554.347,E2 18554.347} C_VEL
LIN {X 0,Y 408.145,Z 468.24,A -85,B 0,C 180,E1 18552.378,E2 18552.378} C_VEL
LIN {X 0,Y 405.942,Z 464.551,A -85,B 0,C 180,E1 18550.789,E2 18550.789} C_VEL
LIN {X 0,Y 402.227,Z 461.955,A -85,B 0,C 180,E1 18547.858,E2 18547.858} C_VEL
LIN {X 0,Y 400.076,Z 458.225,A -85,B 0,C 180,E1 18545.306,E2 18545.306} C_VEL
LIN {X 0,Y 397.54,Z 456.864,A -85,B 0,C 180,E1 18540.576,E2 18540.576} C_VEL
LIN {X 0,Y 397.602,Z 456.864,A -85,B 0,C 180,E1 18535.673,E2 18535.673} C_VEL
LIN {X 0,Y 400.016,Z 458.189,A -85,B 0,C 180,E1 18531.229,E2 18531.229} C_VEL
LIN {X 0,Y 401.219,Z 460.525,A -85,B 0,C 180,E1 18529.663,E2 18529.663} C_VEL
LIN {X 0,Y 403.926,Z 463.5,A -85,B 0,C 180,E1 18527.127,E2 18527.127} C_VEL
LIN {X 0,Y 406.236,Z 464.88,A -85,B 0,C 180,E1 18525.46,E2 18525.46} C_VEL
LIN {X 0,Y 408.369,Z 468.538,A -85,B 0,C 180,E1 18523.938,E2 18523.938} C_VEL
LIN {X 0,Y 411.911,Z 471.405,A -85,B 0,C 180,E1 18521.934,E2 18521.934} C_VEL
LIN {X 0,Y 414.453,Z 475.211,A -85,B 0,C 180,E1 18520.553,E2 18520.553} C_VEL
LIN {X 0,Y 417.443,Z 477.904,A -85,B 0,C 180,E1 18519.164,E2 18519.164} C_VEL
LIN {X 0,Y 420.511,Z 482.022,A -85,B 0,C 180,E1 18517.786,E2 18517.786} C_VEL
LIN {X 0,Y 422.507,Z 483.96,A -85,B 0,C 180,E1 18516.978,E2 18516.978} C_VEL
LIN {X 0,Y 426.026,Z 488.424,A -85,B 0,C 180,E1 18515.595,E2 18515.595} C_VEL
LIN {X 0,Y 427.73,Z 490.409,A -85,B 0,C 180,E1 18514.968,E2 18514.968} C_VEL
LIN {X 0,Y 432.472,Z 496.296,A -85,B 0,C 180,E1 18513.313,E2 18513.313} C_VEL
LIN {X 0,Y 437.213,Z 502.329,A -85,B 0,C 180,E1 18511.782,E2 18511.782} C_VEL
LIN {X 0,Y 444.088,Z 511.094,A -85,B 0,C 180,E1 18509.749,E2 18509.749} C_VEL
LIN {X 0,Y 454.749,Z 525.801,A -85,B 0,C 180,E1 18506.91,E2 18506.91} C_VEL
LIN {X 0,Y 464.273,Z 539.741,A -85,B 0,C 180,E1 18504.634,E2 18504.634} C_VEL
LIN {X 0,Y 474.025,Z 555.052,A -85,B 0,C 180,E1 18502.496,E2 18502.496} C_VEL
LIN {X 0,Y 476.39,Z 559.138,A -85,B 0,C 180,E1 18501.997,E2 18501.997} C_VEL
LIN {X 0,Y 462.776,Z 807.633,A -85,B 0,C 180,E1 18498.045,E2 18498.045} C_VEL
LIN {X 0,Y 460.9,Z 829.692,A -85,B 0,C 180,E1 18497.59,E2 18497.59} C_VEL
LIN {X 0,Y 457.7,Z 855.273,A -85,B 0,C 180,E1 18496.864,E2 18496.864} C_VEL
LIN {X 0,Y 454.561,Z 875.03,A -85,B 0,C 180,E1 18496.14,E2 18496.14} C_VEL
LIN {X 0,Y 450.263,Z 897.956,A -85,B 0,C 180,E1 18495.105,E2 18495.105} C_VEL
LIN {X 0,Y 445.36,Z 919.739,A -85,B 0,C 180,E1 18493.888,E2 18493.888} C_VEL
LIN {X 0,Y 440.17,Z 940.454,A -85,B 0,C 180,E1 18492.517,E2 18492.517} C_VEL
LIN {X 0,Y 434.23,Z 961.434,A -85,B 0,C 180,E1 18490.841,E2 18490.841} C_VEL
LIN {X 0,Y 428.822,Z 979.178,A -85,B 0,C 180,E1 18489.19,E2 18489.19} C_VEL
LIN {X 0,Y 422.192,Z 999.331,A -85,B 0,C 180,E1 18486.982,E2 18486.982} C_VEL
LIN {X 0,Y 416.634,Z 1015.42,A -85,B 0,C 180,E1 18484.917,E2 18484.917} C_VEL
LIN {X 0,Y 410.3,Z 1033.122,A -85,B 0,C 180,E1 18482.256,E2 18482.256} C_VEL
LIN {X 0,Y 405.393,Z 1046.609,A -85,B 0,C 180,E1 18479.883,E2 18479.883} C_VEL
LIN {X 0,Y 400.105,Z 1061.256,A -85,B 0,C 180,E1 18476.894,E2 18476.894} C_VEL
LIN {X 0,Y 395.868,Z 1073.198,A -85,B 0,C 180,E1 18473.995,E2 18473.995} C_VEL
LIN {X 0,Y 392.066,Z 1084.632,A -85,B 0,C 180,E1 18470.763,E2 18470.763} C_VEL
LIN {X 0,Y 389.127,Z 1094.105,A -85,B 0,C 180,E1 18467.496,E2 18467.496} C_VEL
LIN {X 0,Y 387.072,Z 1101.758,A -85,B 0,C 180,E1 18464.359,E2 18464.359} C_VEL
LIN {X 0,Y 385.445,Z 1109.036,A -85,B 0,C 180,E1 18460.614,E2 18460.614} C_VEL
LIN {X 0,Y 384.669,Z 1113.547,A -85,B 0,C 180,E1 18457.618,E2 18457.618} C_VEL
LIN {X 0,Y 384.216,Z 1117.442,A -85,B 0,C 180,E1 18454.179,E2 18454.179} C_VEL
LIN {X 0,Y 384.043,Z 1119.757,A -85,B 0,C 180,E1 18450.746,E2 18450.746} C_VEL
LIN {X 0,Y 384.01,Z 1120.686,A -85,B 0,C 180,E1 18447.762,E2 18447.762} C_VEL
LIN {X 0,Y 384.029,Z 1120.568,A -85,B 0,C 180,E1 18444.622,E2 18444.622} C_VEL
LIN {X 0,Y 384.164,Z 1118.943,A -85,B 0,C 180,E1 18441.016,E2 18441.016} C_VEL
LIN {X 0,Y 384.454,Z 1116.33,A -85,B 0,C 180,E1 18437.934,E2 18437.934} C_VEL
LIN {X 0,Y 385.138,Z 1112.348,A -85,B 0,C 180,E1 18434.644,E2 18434.644} C_VEL
LIN {X 0,Y 386.517,Z 1106.251,A -85,B 0,C 180,E1 18430.977,E2 18430.977} C_VEL
LIN {X 0,Y 388.002,Z 1100.782,A -85,B 0,C 180,E1 18428.333,E2 18428.333} C_VEL
LIN {X 0,Y 387.783,Z 1098.47,A -85,B 0,C 180,E1 18427.242,E2 18427.242} C_VEL
LIN {X 0,Y 384.065,Z 1092.067,A -85,B 0,C 180,E1 18424.282,E2 18424.282} C_VEL
LIN {X 0,Y 384.209,Z 1089.563,A -85,B 0,C 180,E1 18423.358,E2 18423.358} C_VEL
LIN {X 0,Y 387.779,Z 1080.084,A -85,B 0,C 180,E1 18420.325,E2 18420.325} C_VEL
LIN {X 0,Y 392.995,Z 1067.044,A -85,B 0,C 180,E1 18416.832,E2 18416.832} C_VEL
LIN {X 0,Y 397.866,Z 1055.188,A -85,B 0,C 180,E1 18414.157,E2 18414.157} C_VEL
LIN {X 0,Y 404.127,Z 1040.132,A -85,B 0,C 180,E1 18411.246,E2 18411.246} C_VEL
LIN {X 0,Y 410.299,Z 1024.847,A -85,B 0,C 180,E1 18408.755,E2 18408.755} C_VEL
LIN {X 0,Y 417.141,Z 1007.645,A -85,B 0,C 180,E1 18406.343,E2 18406.343} C_VEL
LIN {X 0,Y 423.937,Z 989.333,A -85,B 0,C 180,E1 18404.192,E2 18404.192} C_VEL
LIN {X 0,Y 430.814,Z 969.899,A -85,B 0,C 180,E1 18402.236,E2 18402.236} C_VEL
LIN {X 0,Y 437.33,Z 949.403,A -85,B 0,C 180,E1 18400.517,E2 18400.517} C_VEL
LIN {X 0,Y 443.17,Z 929.427,A -85,B 0,C 180,E1 18399.091,E2 18399.091} C_VEL
LIN {X 0,Y 448.976,Z 906.778,A -85,B 0,C 180,E1 18397.758,E2 18397.758} C_VEL
LIN {X 0,Y 453.296,Z 887.358,A -85,B 0,C 180,E1 18396.801,E2 18396.801} C_VEL
LIN {X 0,Y 458.051,Z 861.985,A -85,B 0,C 180,E1 18395.796,E2 18395.796} C_VEL
LIN {X 0,Y 461.246,Z 840.4,A -85,B 0,C 180,E1 18395.134,E2 18395.134} C_VEL
LIN {X 0,Y 464.065,Z 814.855,A -85,B 0,C 180,E1 18394.549,E2 18394.549} C_VEL
LIN {X 0,Y 469.019,Z 734.55,A -85,B 0,C 180,E1 18393.249,E2 18393.249} C_VEL
LIN {X 0,Y 479.123,Z 567.549,A -85,B 0,C 180,E1 18390.594,E2 18390.594} C_VEL
LIN {X 0,Y 469.62,Z 552.705,A -85,B 0,C 180,E1 18388.243,E2 18388.243} C_VEL
LIN {X 0,Y 459.319,Z 537.714,A -85,B 0,C 180,E1 18385.395,E2 18385.395} C_VEL
LIN {X 0,Y 450.93,Z 526.225,A -85,B 0,C 180,E1 18382.764,E2 18382.764} C_VEL
LIN {X 0,Y 445.268,Z 519.009,A -85,B 0,C 180,E1 18380.782,E2 18380.782} C_VEL
LIN {X 0,Y 442.232,Z 515.057,A -85,B 0,C 180,E1 18379.619,E2 18379.619} C_VEL
LIN {X 0,Y 438.185,Z 509.891,A -85,B 0,C 180,E1 18377.942,E2 18377.942} C_VEL
LIN {X 0,Y 434.481,Z 505.081,A -85,B 0,C 180,E1 18376.237,E2 18376.237} C_VEL
LIN {X 0,Y 430.58,Z 500.656,A -85,B 0,C 180,E1 18374.25,E2 18374.25} C_VEL
LIN {X 0,Y 429.474,Z 498.895,A -85,B 0,C 180,E1 18373.6,E2 18373.6} C_VEL
LIN {X 0,Y 426.228,Z 495.829,A -85,B 0,C 180,E1 18371.639,E2 18371.639} C_VEL
LIN {X 0,Y 424.463,Z 492.797,A -85,B 0,C 180,E1 18370.313,E2 18370.313} C_VEL
LIN {X 0,Y 421.348,Z 490.32,A -85,B 0,C 180,E1 18367.774,E2 18367.774} C_VEL
LIN {X 0,Y 419.346,Z 486.569,A -85,B 0,C 180,E1 18365.336,E2 18365.336} C_VEL
LIN {X 0,Y 416.732,Z 485.152,A -85,B 0,C 180,E1 18359.038,E2 18359.038} C_VEL
LIN {X 0,Y 418.241,Z 486.061,A -85,B 0,C 180,E1 18353.686,E2 18353.686} C_VEL
LIN {X 0,Y 419.61,Z 486.887,A -85,B 0,C 180,E1 18351.78,E2 18351.78} C_VEL
LIN {X 0,Y 421.429,Z 490.4,A -85,B 0,C 180,E1 18349.612,E2 18349.612} C_VEL
LIN {X 0,Y 424.83,Z 493.297,A -85,B 0,C 180,E1 18346.872,E2 18346.872} C_VEL
LIN {X 0,Y 427.403,Z 497.186,A -85,B 0,C 180,E1 18345.061,E2 18345.061} C_VEL
LIN {X 0,Y 429.835,Z 499.408,A -85,B 0,C 180,E1 18343.652,E2 18343.652} C_VEL
LIN {X 0,Y 433.053,Z 503.736,A -85,B 0,C 180,E1 18341.907,E2 18341.907} C_VEL
LIN {X 0,Y 434.771,Z 505.58,A -85,B 0,C 180,E1 18341.078,E2 18341.078} C_VEL
LIN {X 0,Y 441,Z 514.128,A -85,B 0,C 180,E1 18338.311,E2 18338.311} C_VEL
LIN {X 0,Y 447.892,Z 524.029,A -85,B 0,C 180,E1 18335.677,E2 18335.677} C_VEL
LIN {X 0,Y 457.022,Z 537.883,A -85,B 0,C 180,E1 18332.648,E2 18332.648} C_VEL
LIN {X 0,Y 466.695,Z 553.572,A -85,B 0,C 180,E1 18329.84,E2 18329.84} C_VEL
LIN {X 0,Y 475.889,Z 569.72,A -85,B 0,C 180,E1 18327.442,E2 18327.442} C_VEL
LIN {X 0,Y 478.917,Z 575.643,A -85,B 0,C 180,E1 18326.691,E2 18326.691} C_VEL
LIN {X 0,Y 465.864,Z 793.41,A -85,B 0,C 180,E1 18323.224,E2 18323.224} C_VEL
LIN {X 0,Y 462.967,Z 838.019,A -85,B 0,C 180,E1 18322.482,E2 18322.482} C_VEL
LIN {X 0,Y 459.975,Z 862.339,A -85,B 0,C 180,E1 18321.928,E2 18321.928} C_VEL
LIN {X 0,Y 456.064,Z 886.595,A -85,B 0,C 180,E1 18321.207,E2 18321.207} C_VEL
LIN {X 0,Y 451.442,Z 909.145,A -85,B 0,C 180,E1 18320.325,E2 18320.325} C_VEL
LIN {X 0,Y 446.453,Z 930.475,A -85,B 0,C 180,E1 18319.299,E2 18319.299} C_VEL
LIN {X 0,Y 440.244,Z 953.524,A -85,B 0,C 180,E1 18317.932,E2 18317.932} C_VEL
LIN {X 0,Y 434.447,Z 972.848,A -85,B 0,C 180,E1 18316.563,E2 18316.563} C_VEL
LIN {X 0,Y 427.235,Z 994.911,A -85,B 0,C 180,E1 18314.691,E2 18314.691} C_VEL
LIN {X 0,Y 420.909,Z 1012.825,A -85,B 0,C 180,E1 18312.891,E2 18312.891} C_VEL
LIN {X 0,Y 413.617,Z 1032.481,A -85,B 0,C 180,E1 18310.564,E2 18310.564} C_VEL
LIN {X 0,Y 407.519,Z 1048.189,A -85,B 0,C 180,E1 18308.372,E2 18308.372} C_VEL
LIN {X 0,Y 401.032,Z 1064.769,A -85,B 0,C 180,E1 18305.692,E2 18305.692} C_VEL
LIN {X 0,Y 395.073,Z 1079.801,A -85,B 0,C 180,E1 18302.794,E2 18302.794} C_VEL
LIN {X 0,Y 389.798,Z 1093.686,A -85,B 0,C 180,E1 18299.675,E2 18299.675} C_VEL
LIN {X 0,Y 385.469,Z 1105.484,A -85,B 0,C 180,E1 18296.498,E2 18296.498} C_VEL
LIN {X 0,Y 382.076,Z 1115.734,A -85,B 0,C 180,E1 18293.276,E2 18293.276} C_VEL
LIN {X 0,Y 379.265,Z 1125.45,A -85,B 0,C 180,E1 18289.562,E2 18289.562} C_VEL
LIN {X 0,Y 377.627,Z 1132.453,A -85,B 0,C 180,E1 18286.3,E2 18286.3} C_VEL
LIN {X 0,Y 376.493,Z 1139.015,A -85,B 0,C 180,E1 18282.423,E2 18282.423} C_VEL
LIN {X 0,Y 376.08,Z 1143.07,A -85,B 0,C 180,E1 18279.179,E2 18279.179} C_VEL
LIN {X 0,Y 375.981,Z 1145.923,A -85,B 0,C 180,E1 18275.942,E2 18275.942} C_VEL
LIN {X 0,Y 375.992,Z 1147.571,A -85,B 0,C 180,E1 18272.439,E2 18272.439} C_VEL
LIN {X 0,Y 376.005,Z 1147.761,A -85,B 0,C 180,E1 18269.391,E2 18269.391} C_VEL
LIN {X 0,Y 375.996,Z 1146.922,A -85,B 0,C 180,E1 18266.493,E2 18266.493} C_VEL
LIN {X 0,Y 375.998,Z 1144.956,A -85,B 0,C 180,E1 18263.434,E2 18263.434} C_VEL
LIN {X 0,Y 376.18,Z 1141.065,A -85,B 0,C 180,E1 18259.742,E2 18259.742} C_VEL
LIN {X 0,Y 376.718,Z 1136.206,A -85,B 0,C 180,E1 18256.493,E2 18256.493} C_VEL
LIN {X 0,Y 377.826,Z 1129.748,A -85,B 0,C 180,E1 18253.076,E2 18253.076} C_VEL
LIN {X 0,Y 379.748,Z 1121.217,A -85,B 0,C 180,E1 18249.501,E2 18249.501} C_VEL
LIN {X 0,Y 382.165,Z 1112.348,A -85,B 0,C 180,E1 18246.403,E2 18246.403} C_VEL
LIN {X 0,Y 386.103,Z 1099.72,A -85,B 0,C 180,E1 18242.717,E2 18242.717} C_VEL
LIN {X 0,Y 390.066,Z 1088.003,A -85,B 0,C 180,E1 18239.839,E2 18239.839} C_VEL
LIN {X 0,Y 395.365,Z 1073.134,A -85,B 0,C 180,E1 18236.715,E2 18236.715} C_VEL
LIN {X 0,Y 400.677,Z 1058.419,A -85,B 0,C 180,E1 18234.095,E2 18234.095} C_VEL
LIN {X 0,Y 406.892,Z 1041.308,A -85,B 0,C 180,E1 18231.468,E2 18231.468} C_VEL
LIN {X 0,Y 413.053,Z 1023.693,A -85,B 0,C 180,E1 18229.186,E2 18229.186} C_VEL
LIN {X 0,Y 419.631,Z 1004.413,A -85,B 0,C 180,E1 18227.041,E2 18227.041} C_VEL
LIN {X 0,Y 425.812,Z 984.813,A -85,B 0,C 180,E1 18225.214,E2 18225.214} C_VEL
LIN {X 0,Y 431.691,Z 964.988,A -85,B 0,C 180,E1 18223.629,E2 18223.629} C_VEL
LIN {X 0,Y 437.656,Z 942.668,A -85,B 0,C 180,E1 18222.152,E2 18222.152} C_VEL
LIN {X 0,Y 442.406,Z 922.744,A -85,B 0,C 180,E1 18221.045,E2 18221.045} C_VEL
LIN {X 0,Y 447.565,Z 897.89,A -85,B 0,C 180,E1 18219.928,E2 18219.928} C_VEL
LIN {X 0,Y 451.278,Z 876.456,A -85,B 0,C 180,E1 18219.169,E2 18219.169} C_VEL
LIN {X 0,Y 454.851,Z 850.438,A -85,B 0,C 180,E1 18218.467,E2 18218.467} C_VEL
LIN {X 0,Y 456.876,Z 827.924,A -85,B 0,C 180,E1 18218.016,E2 18218.016} C_VEL
LIN {X 0,Y 469.248,Z 604.875,A -85,B 0,C 180,E1 18214.437,E2 18214.437} C_VEL
LIN {X 0,Y 471.112,Z 570.623,A -85,B 0,C 180,E1 18213.876,E2 18213.876} C_VEL
LIN {X 0,Y 461.549,Z 553.061,A -85,B 0,C 180,E1 18211.692,E2 18211.692} C_VEL
LIN {X 0,Y 452.729,Z 538.119,A -85,B 0,C 180,E1 18209.506,E2 18209.506} C_VEL
LIN {X 0,Y 444.615,Z 525.186,A -85,B 0,C 180,E1 18207.308,E2 18207.308} C_VEL
LIN {X 0,Y 437.025,Z 513.635,A -85,B 0,C 180,E1 18205.041,E2 18205.041} C_VEL
LIN {X 0,Y 429.35,Z 502.705,A -85,B 0,C 180,E1 18202.49,E2 18202.49} C_VEL
LIN {X 0,Y 424.468,Z 496.13,A -85,B 0,C 180,E1 18200.692,E2 18200.692} C_VEL
LIN {X 0,Y 420.675,Z 491.458,A -85,B 0,C 180,E1 18199.184,E2 18199.184} C_VEL
LIN {X 0,Y 416.179,Z 486.232,A -85,B 0,C 180,E1 18197.224,E2 18197.224} C_VEL
LIN {X 0,Y 415.003,Z 484.674,A -85,B 0,C 180,E1 18196.661,E2 18196.661} C_VEL
LIN {X 0,Y 411.637,Z 481.272,A -85,B 0,C 180,E1 18194.993,E2 18194.993} C_VEL
LIN {X 0,Y 410.12,Z 478.713,A -85,B 0,C 180,E1 18194.111,E2 18194.111} C_VEL
LIN {X 0,Y 406.637,Z 475.788,A -85,B 0,C 180,E1 18192.064,E2 18192.064} C_VEL
LIN {X 0,Y 404.774,Z 472.435,A -85,B 0,C 180,E1 18190.677,E2 18190.677} C_VEL
LIN {X 0,Y 401.102,Z 469.837,A -85,B 0,C 180,E1 18187.736,E2 18187.736} C_VEL
LIN {X 0,Y 398.99,Z 466.103,A -85,B 0,C 180,E1 18185.176,E2 18185.176} C_VEL
LIN {X 0,Y 396.432,Z 464.71,A -85,B 0,C 180,E1 18180,E2 18180} C_VEL
LIN {X 0,Y 396.762,Z 464.907,A -85,B 0,C 180,E1 18175.229,E2 18175.229} C_VEL
LIN {X 0,Y 399.044,Z 466.191,A -85,B 0,C 180,E1 18171.208,E2 18171.208} C_VEL
LIN {X 0,Y 401.478,Z 470.293,A -85,B 0,C 180,E1 18168.362,E2 18168.362} C_VEL
LIN {X 0,Y 404.913,Z 472.778,A -85,B 0,C 180,E1 18165.667,E2 18165.667} C_VEL
LIN {X 0,Y 407.186,Z 476.482,A -85,B 0,C 180,E1 18164.036,E2 18164.036} C_VEL
LIN {X 0,Y 410.383,Z 479.138,A -85,B 0,C 180,E1 18162.195,E2 18162.195} C_VEL
LIN {X 0,Y 413.227,Z 483.185,A -85,B 0,C 180,E1 18160.64,E2 18160.64} C_VEL
LIN {X 0,Y 415.756,Z 485.543,A -85,B 0,C 180,E1 18159.443,E2 18159.443} C_VEL
LIN {X 0,Y 419.097,Z 489.872,A -85,B 0,C 180,E1 18157.928,E2 18157.928} C_VEL
LIN {X 0,Y 420.743,Z 491.616,A -85,B 0,C 180,E1 18157.246,E2 18157.246} C_VEL
LIN {X 0,Y 424.555,Z 496.28,A -85,B 0,C 180,E1 18155.734,E2 18155.734} C_VEL
LIN {X 0,Y 430.314,Z 503.582,A -85,B 0,C 180,E1 18153.652,E2 18153.652} C_VEL
LIN {X 0,Y 435.372,Z 510.135,A -85,B 0,C 180,E1 18151.987,E2 18151.987} C_VEL
LIN {X 0,Y 441.769,Z 518.451,A -85,B 0,C 180,E1 18150.061,E2 18150.061} C_VEL
LIN {X 0,Y 451.842,Z 532.521,A -85,B 0,C 180,E1 18147.319,E2 18147.319} C_VEL
LIN {X 0,Y 461.131,Z 546.313,A -85,B 0,C 180,E1 18145.045,E2 18145.045} C_VEL
LIN {X 0,Y 470.77,Z 561.685,A -85,B 0,C 180,E1 18142.881,E2 18142.881} C_VEL
LIN {X 0,Y 471.476,Z 563.21,A -85,B 0,C 180,E1 18142.72,E2 18142.72} C_VEL
LIN {X 0,Y 457.608,Z 808.462,A -85,B 0,C 180,E1 18138.799,E2 18138.799} C_VEL
LIN {X 0,Y 455.628,Z 830.925,A -85,B 0,C 180,E1 18138.331,E2 18138.331} C_VEL
LIN {X 0,Y 452.388,Z 855.89,A -85,B 0,C 180,E1 18137.613,E2 18137.613} C_VEL
LIN {X 0,Y 449.187,Z 875.487,A -85,B 0,C 180,E1 18136.891,E2 18136.891} C_VEL
LIN {X 0,Y 444.679,Z 898.776,A -85,B 0,C 180,E1 18135.832,E2 18135.832} C_VEL
LIN {X 0,Y 439.993,Z 919.079,A -85,B 0,C 180,E1 18134.696,E2 18134.696} C_VEL
LIN {X 0,Y 434.786,Z 939.311,A -85,B 0,C 180,E1 18133.361,E2 18133.361} C_VEL
LIN {X 0,Y 428.639,Z 960.626,A -85,B 0,C 180,E1 18131.669,E2 18131.669} C_VEL
LIN {X 0,Y 423.036,Z 978.473,A -85,B 0,C 180,E1 18130.009,E2 18130.009} C_VEL
LIN {X 0,Y 416.126,Z 998.944,A -85,B 0,C 180,E1 18127.764,E2 18127.764} C_VEL
LIN {X 0,Y 410.399,Z 1014.961,A -85,B 0,C 180,E1 18125.698,E2 18125.698} C_VEL
LIN {X 0,Y 403.794,Z 1032.789,A -85,B 0,C 180,E1 18123.009,E2 18123.009} C_VEL
LIN {X 0,Y 398.385,Z 1047.086,A -85,B 0,C 180,E1 18120.464,E2 18120.464} C_VEL
LIN {X 0,Y 392.888,Z 1061.701,A -85,B 0,C 180,E1 18117.429,E2 18117.429} C_VEL
LIN {X 0,Y 388.467,Z 1073.629,A -85,B 0,C 180,E1 18114.482,E2 18114.482} C_VEL
LIN {X 0,Y 384.495,Z 1085.039,A -85,B 0,C 180,E1 18111.191,E2 18111.191} C_VEL
LIN {X 0,Y 381.415,Z 1094.493,A -85,B 0,C 180,E1 18107.862,E2 18107.862} C_VEL
LIN {X 0,Y 379.167,Z 1102.477,A -85,B 0,C 180,E1 18104.508,E2 18104.508} C_VEL
LIN {X 0,Y 377.53,Z 1109.386,A -85,B 0,C 180,E1 18100.839,E2 18100.839} C_VEL
LIN {X 0,Y 376.684,Z 1114.085,A -85,B 0,C 180,E1 18097.627,E2 18097.627} C_VEL
LIN {X 0,Y 376.201,Z 1118.005,A -85,B 0,C 180,E1 18093.963,E2 18093.963} C_VEL
LIN {X 0,Y 376.052,Z 1120.125,A -85,B 0,C 180,E1 18090.609,E2 18090.609} C_VEL
LIN {X 0,Y 376.013,Z 1120.999,A -85,B 0,C 180,E1 18087.561,E2 18087.561} C_VEL
LIN {X 0,Y 376.059,Z 1120.736,A -85,B 0,C 180,E1 18083.945,E2 18083.945} C_VEL
LIN {X 0,Y 376.19,Z 1118.982,A -85,B 0,C 180,E1 18080.515,E2 18080.515} C_VEL
LIN {X 0,Y 376.537,Z 1116.326,A -85,B 0,C 180,E1 18077.423,E2 18077.423} C_VEL
LIN {X 0,Y 377.447,Z 1111.709,A -85,B 0,C 180,E1 18073.692,E2 18073.692} C_VEL
LIN {X 0,Y 378.885,Z 1105.873,A -85,B 0,C 180,E1 18070.257,E2 18070.257} C_VEL
LIN {X 0,Y 381.207,Z 1098.301,A -85,B 0,C 180,E1 18066.667,E2 18066.667} C_VEL
LIN {X 0,Y 384.209,Z 1089.563,A -85,B 0,C 180,E1 18063.358,E2 18063.358} C_VEL
LIN {X 0,Y 384.354,Z 1086.662,A -85,B 0,C 180,E1 18062.285,E2 18062.285} C_VEL
LIN {X 0,Y 381.823,Z 1078.913,A -85,B 0,C 180,E1 18059.349,E2 18059.349} C_VEL
LIN {X 0,Y 382.355,Z 1075.95,A -85,B 0,C 180,E1 18058.457,E2 18058.457} C_VEL
LIN {X 0,Y 387.116,Z 1064.675,A -85,B 0,C 180,E1 18055.552,E2 18055.552} C_VEL
LIN {X 0,Y 393.065,Z 1050.972,A -85,B 0,C 180,E1 18052.531,E2 18052.531} C_VEL
LIN {X 0,Y 399.421,Z 1036.006,A -85,B 0,C 180,E1 18049.769,E2 18049.769} C_VEL
LIN {X 0,Y 406.465,Z 1019.368,A -85,B 0,C 180,E1 18047.145,E2 18047.145} C_VEL
LIN {X 0,Y 413.338,Z 1002.118,A -85,B 0,C 180,E1 18044.864,E2 18044.864} C_VEL
LIN {X 0,Y 420.215,Z 984.151,A -85,B 0,C 180,E1 18042.821,E2 18042.821} C_VEL
LIN {X 0,Y 427.277,Z 963.968,A -85,B 0,C 180,E1 18040.898,E2 18040.898} C_VEL
LIN {X 0,Y 433.336,Z 945.231,A -85,B 0,C 180,E1 18039.377,E2 18039.377} C_VEL
LIN {X 0,Y 439.763,Z 923.044,A -85,B 0,C 180,E1 18037.872,E2 18037.872} C_VEL
LIN {X 0,Y 444.584,Z 904.25,A -85,B 0,C 180,E1 18036.806,E2 18036.806} C_VEL
LIN {X 0,Y 449.631,Z 881.784,A -85,B 0,C 180,E1 18035.738,E2 18035.738} C_VEL
LIN {X 0,Y 453.699,Z 859.37,A -85,B 0,C 180,E1 18034.897,E2 18034.897} C_VEL
LIN {X 0,Y 456.974,Z 837.329,A -85,B 0,C 180,E1 18034.24,E2 18034.24} C_VEL
LIN {X 0,Y 459.609,Z 812.208,A -85,B 0,C 180,E1 18033.692,E2 18033.692} C_VEL
LIN {X 0,Y 473.796,Z 585.902,A -85,B 0,C 180,E1 18030.074,E2 18030.074} C_VEL
LIN {X 0,Y 474.675,Z 571.878,A -85,B 0,C 180,E1 18029.849,E2 18029.849} C_VEL
LIN {X 0,Y 465.859,Z 558.007,A -85,B 0,C 180,E1 18027.586,E2 18027.586} C_VEL
LIN {X 0,Y 455.628,Z 542.905,A -85,B 0,C 180,E1 18024.643,E2 18024.643} C_VEL
LIN {X 0,Y 447.641,Z 532.113,A -85,B 0,C 180,E1 18022.04,E2 18022.04} C_VEL
LIN {X 0,Y 443.462,Z 526.569,A -85,B 0,C 180,E1 18020.525,E2 18020.525} C_VEL
LIN {X 0,Y 440.157,Z 522.247,A -85,B 0,C 180,E1 18019.232,E2 18019.232} C_VEL
LIN {X 0,Y 436.337,Z 517.289,A -85,B 0,C 180,E1 18017.607,E2 18017.607} C_VEL
LIN {X 0,Y 432.176,Z 512.015,A -85,B 0,C 180,E1 18015.637,E2 18015.637} C_VEL
LIN {X 0,Y 428.689,Z 507.645,A -85,B 0,C 180,E1 18013.763,E2 18013.763} C_VEL
LIN {X 0,Y 427.806,Z 506.466,A -85,B 0,C 180,E1 18013.241,E2 18013.241} C_VEL
LIN {X 0,Y 424.673,Z 503.234,A -85,B 0,C 180,E1 18011.27,E2 18011.27} C_VEL
LIN {X 0,Y 423.124,Z 500.577,A -85,B 0,C 180,E1 18010.071,E2 18010.071} C_VEL
LIN {X 0,Y 420.099,Z 498.023,A -85,B 0,C 180,E1 18007.522,E2 18007.522} C_VEL
LIN {X 0,Y 418.266,Z 494.46,A -85,B 0,C 180,E1 18005.212,E2 18005.212} C_VEL
LIN {X 0,Y 415.754,Z 493.083,A -85,B 0,C 180,E1 17998.898,E2 17998.898} C_VEL
LIN {X 0,Y 417.626,Z 494.16,A -85,B 0,C 180,E1 17993.125,E2 17993.125} C_VEL
LIN {X 0,Y 418.521,Z 494.85,A -85,B 0,C 180,E1 17991.897,E2 17991.897} C_VEL
LIN {X 0,Y 420.456,Z 498.453,A -85,B 0,C 180,E1 17989.587,E2 17989.587} C_VEL
LIN {X 0,Y 423.496,Z 501.026,A -85,B 0,C 180,E1 17987.108,E2 17987.108} C_VEL
LIN {X 0,Y 426.187,Z 505.059,A -85,B 0,C 180,E1 17985.183,E2 17985.183} C_VEL
LIN {X 0,Y 428.401,Z 507.166,A -85,B 0,C 180,E1 17983.874,E2 17983.874} C_VEL
LIN {X 0,Y 431.705,Z 511.553,A -85,B 0,C 180,E1 17982.058,E2 17982.058} C_VEL
LIN {X 0,Y 433.262,Z 513.357,A -85,B 0,C 180,E1 17981.289,E2 17981.289} C_VEL
LIN {X 0,Y 439.109,Z 521.521,A -85,B 0,C 180,E1 17978.633,E2 17978.633} C_VEL
LIN {X 0,Y 445.721,Z 531.181,A -85,B 0,C 180,E1 17976.044,E2 17976.044} C_VEL
LIN {X 0,Y 454.605,Z 544.925,A -85,B 0,C 180,E1 17973.022,E2 17973.022} C_VEL
LIN {X 0,Y 464.231,Z 560.831,A -85,B 0,C 180,E1 17970.162,E2 17970.162} C_VEL
LIN {X 0,Y 472.867,Z 576.352,A -85,B 0,C 180,E1 17967.855,E2 17967.855} C_VEL
LIN {X 0,Y 474.434,Z 579.668,A -85,B 0,C 180,E1 17967.447,E2 17967.447} C_VEL
LIN {X 0,Y 461.008,Z 797.17,A -85,B 0,C 180,E1 17963.973,E2 17963.973} C_VEL
LIN {X 0,Y 458.218,Z 838.175,A -85,B 0,C 180,E1 17963.284,E2 17963.284} C_VEL
LIN {X 0,Y 455.181,Z 862.23,A -85,B 0,C 180,E1 17962.735,E2 17962.735} C_VEL
LIN {X 0,Y 451.262,Z 885.979,A -85,B 0,C 180,E1 17962.032,E2 17962.032} C_VEL
LIN {X 0,Y 446.356,Z 909.338,A -85,B 0,C 180,E1 17961.118,E2 17961.118} C_VEL
LIN {X 0,Y 440.967,Z 931.738,A -85,B 0,C 180,E1 17960.033,E2 17960.033} C_VEL
LIN {X 0,Y 434.708,Z 954.092,A -85,B 0,C 180,E1 17958.689,E2 17958.689} C_VEL
LIN {X 0,Y 428.651,Z 973.676,A -85,B 0,C 180,E1 17957.289,E2 17957.289} C_VEL
LIN {X 0,Y 421.231,Z 995.54,A -85,B 0,C 180,E1 17955.408,E2 17955.408} C_VEL
LIN {X 0,Y 414.72,Z 1013.37,A -85,B 0,C 180,E1 17953.594,E2 17953.594} C_VEL
LIN {X 0,Y 406.991,Z 1033.394,A -85,B 0,C 180,E1 17951.18,E2 17951.18} C_VEL
LIN {X 0,Y 400.711,Z 1048.999,A -85,B 0,C 180,E1 17948.963,E2 17948.963} C_VEL
LIN {X 0,Y 393.674,Z 1066.172,A -85,B 0,C 180,E1 17946.104,E2 17946.104} C_VEL
LIN {X 0,Y 387.846,Z 1080.342,A -85,B 0,C 180,E1 17943.307,E2 17943.307} C_VEL
LIN {X 0,Y 382.134,Z 1094.658,A -85,B 0,C 180,E1 17939.985,E2 17939.985} C_VEL
LIN {X 0,Y 377.875,Z 1105.805,A -85,B 0,C 180,E1 17936.903,E2 17936.903} C_VEL
LIN {X 0,Y 374.202,Z 1116.452,A -85,B 0,C 180,E1 17933.462,E2 17933.462} C_VEL
LIN {X 0,Y 371.409,Z 1125.58,A -85,B 0,C 180,E1 17929.829,E2 17929.829} C_VEL
LIN {X 0,Y 369.633,Z 1132.835,A -85,B 0,C 180,E1 17926.34,E2 17926.34} C_VEL
LIN {X 0,Y 368.513,Z 1138.974,A -85,B 0,C 180,E1 17922.537,E2 17922.537} C_VEL
LIN {X 0,Y 368.094,Z 1142.809,A -85,B 0,C 180,E1 17919.38,E2 17919.38} C_VEL
LIN {X 0,Y 367.984,Z 1145.703,A -85,B 0,C 180,E1 17916.009,E2 17916.009} C_VEL
LIN {X 0,Y 367.994,Z 1147.29,A -85,B 0,C 180,E1 17912.492,E2 17912.492} C_VEL
LIN {X 0,Y 368.011,Z 1147.473,A -85,B 0,C 180,E1 17909.377,E2 17909.377} C_VEL
LIN {X 0,Y 368.002,Z 1146.626,A -85,B 0,C 180,E1 17906.417,E2 17906.417} C_VEL
LIN {X 0,Y 368.005,Z 1144.65,A -85,B 0,C 180,E1 17903.291,E2 17903.291} C_VEL
LIN {X 0,Y 368.201,Z 1140.741,A -85,B 0,C 180,E1 17899.517,E2 17899.517} C_VEL
LIN {X 0,Y 368.785,Z 1135.871,A -85,B 0,C 180,E1 17896.196,E2 17896.196} C_VEL
LIN {X 0,Y 370.042,Z 1129.089,A -85,B 0,C 180,E1 17892.546,E2 17892.546} C_VEL
LIN {X 0,Y 372.122,Z 1120.434,A -85,B 0,C 180,E1 17888.896,E2 17888.896} C_VEL
LIN {X 0,Y 374.737,Z 1111.5,A -85,B 0,C 180,E1 17885.738,E2 17885.738} C_VEL
LIN {X 0,Y 378.735,Z 1099.319,A -85,B 0,C 180,E1 17882.141,E2 17882.141} C_VEL
LIN {X 0,Y 382.887,Z 1087.59,A -85,B 0,C 180,E1 17879.213,E2 17879.213} C_VEL
LIN {X 0,Y 388.626,Z 1072.173,A -85,B 0,C 180,E1 17875.942,E2 17875.942} C_VEL
LIN {X 0,Y 393.968,Z 1057.966,A -85,B 0,C 180,E1 17873.385,E2 17873.385} C_VEL
LIN {X 0,Y 400.443,Z 1040.769,A -85,B 0,C 180,E1 17870.72,E2 17870.72} C_VEL
LIN {X 0,Y 406.821,Z 1023.189,A -85,B 0,C 180,E1 17868.424,E2 17868.424} C_VEL
LIN {X 0,Y 413.63,Z 1003.869,A -85,B 0,C 180,E1 17866.262,E2 17866.262} C_VEL
LIN {X 0,Y 420.038,Z 984.165,A -85,B 0,C 180,E1 17864.416,E2 17864.416} C_VEL
LIN {X 0,Y 426.333,Z 963.567,A -85,B 0,C 180,E1 17862.769,E2 17862.769} C_VEL
LIN {X 0,Y 432.231,Z 941.919,A -85,B 0,C 180,E1 17861.343,E2 17861.343} C_VEL
LIN {X 0,Y 437.065,Z 922.167,A -85,B 0,C 180,E1 17860.247,E2 17860.247} C_VEL
LIN {X 0,Y 442.254,Z 897.789,A -85,B 0,C 180,E1 17859.15,E2 17859.15} C_VEL
LIN {X 0,Y 446.048,Z 876.444,A -85,B 0,C 180,E1 17858.392,E2 17858.392} C_VEL
LIN {X 0,Y 449.676,Z 850.847,A -85,B 0,C 180,E1 17857.696,E2 17857.696} C_VEL
LIN {X 0,Y 451.792,Z 828.071,A -85,B 0,C 180,E1 17857.235,E2 17857.235} C_VEL
LIN {X 0,Y 464.529,Z 605.643,A -85,B 0,C 180,E1 17853.649,E2 17853.649} C_VEL
LIN {X 0,Y 466.283,Z 574.232,A -85,B 0,C 180,E1 17853.131,E2 17853.131} C_VEL
LIN {X 0,Y 456.583,Z 556.413,A -85,B 0,C 180,E1 17850.827,E2 17850.827} C_VEL
LIN {X 0,Y 447.151,Z 540.341,A -85,B 0,C 180,E1 17848.371,E2 17848.371} C_VEL
LIN {X 0,Y 439.126,Z 527.661,A -85,B 0,C 180,E1 17846.07,E2 17846.07} C_VEL
LIN {X 0,Y 431.68,Z 516.362,A -85,B 0,C 180,E1 17843.696,E2 17843.696} C_VEL
LIN {X 0,Y 425.064,Z 506.927,A -85,B 0,C 180,E1 17841.348,E2 17841.348} C_VEL
LIN {X 0,Y 422.148,Z 503.181,A -85,B 0,C 180,E1 17840.231,E2 17840.231} C_VEL
LIN {X 0,Y 417.912,Z 497.883,A -85,B 0,C 180,E1 17838.483,E2 17838.483} C_VEL
LIN {X 0,Y 414.284,Z 493.476,A -85,B 0,C 180,E1 17836.836,E2 17836.836} C_VEL
LIN {X 0,Y 413.184,Z 492.163,A -85,B 0,C 180,E1 17836.303,E2 17836.303} C_VEL
LIN {X 0,Y 409.791,Z 488.442,A -85,B 0,C 180,E1 17834.556,E2 17834.556} C_VEL
LIN {X 0,Y 408.406,Z 486.301,A -85,B 0,C 180,E1 17833.738,E2 17833.738} C_VEL
LIN {X 0,Y 405.041,Z 483.196,A -85,B 0,C 180,E1 17831.679,E2 17831.679} C_VEL
LIN {X 0,Y 403.406,Z 480.234,A -85,B 0,C 180,E1 17830.425,E2 17830.425} C_VEL
LIN {X 0,Y 399.838,Z 477.544,A -85,B 0,C 180,E1 17827.472,E2 17827.472} C_VEL
LIN {X 0,Y 397.8,Z 473.892,A -85,B 0,C 180,E1 17824.903,E2 17824.903} C_VEL
LIN {X 0,Y 395.316,Z 472.536,A -85,B 0,C 180,E1 17818.985,E2 17818.985} C_VEL
LIN {X 0,Y 396.713,Z 473.302,A -85,B 0,C 180,E1 17813.197,E2 17813.197} C_VEL
LIN {X 0,Y 398.068,Z 474.231,A -85,B 0,C 180,E1 17811.186,E2 17811.186} C_VEL
LIN {X 0,Y 400.21,Z 478.027,A -85,B 0,C 180,E1 17808.616,E2 17808.616} C_VEL
LIN {X 0,Y 403.516,Z 480.454,A -85,B 0,C 180,E1 17805.946,E2 17805.946} C_VEL
LIN {X 0,Y 406.004,Z 484.417,A -85,B 0,C 180,E1 17804.135,E2 17804.135} C_VEL
LIN {X 0,Y 408.921,Z 486.954,A -85,B 0,C 180,E1 17802.423,E2 17802.423} C_VEL
LIN {X 0,Y 411.817,Z 490.963,A -85,B 0,C 180,E1 17800.821,E2 17800.821} C_VEL
LIN {X 0,Y 414.082,Z 493.161,A -85,B 0,C 180,E1 17799.726,E2 17799.726} C_VEL
LIN {X 0,Y 417.531,Z 497.572,A -85,B 0,C 180,E1 17798.137,E2 17798.137} C_VEL
LIN {X 0,Y 419.065,Z 499.369,A -85,B 0,C 180,E1 17797.483,E2 17797.483} C_VEL
LIN {X 0,Y 423.911,Z 505.457,A -85,B 0,C 180,E1 17795.546,E2 17795.546} C_VEL
LIN {X 0,Y 428.349,Z 511.119,A -85,B 0,C 180,E1 17793.932,E2 17793.932} C_VEL
LIN {X 0,Y 435.584,Z 520.478,A -85,B 0,C 180,E1 17791.554,E2 17791.554} C_VEL
LIN {X 0,Y 445.517,Z 534.217,A -85,B 0,C 180,E1 17788.659,E2 17788.659} C_VEL
LIN {X 0,Y 456.652,Z 550.68,A -85,B 0,C 180,E1 17785.793,E2 17785.793} C_VEL
LIN {X 0,Y 466.584,Z 566.693,A -85,B 0,C 180,E1 17783.484,E2 17783.484} C_VEL
LIN {X 0,Y 455.544,Z 757.95,A -85,B 0,C 180,E1 17780.411,E2 17780.411} C_VEL
LIN {X 0,Y 452.014,Z 816.229,A -85,B 0,C 180,E1 17779.446,E2 17779.446} C_VEL
LIN {X 0,Y 449.291,Z 841.058,A -85,B 0,C 180,E1 17778.855,E2 17778.855} C_VEL
LIN {X 0,Y 446.059,Z 863.466,A -85,B 0,C 180,E1 17778.146,E2 17778.146} C_VEL
LIN {X 0,Y 441.713,Z 887.234,A -85,B 0,C 180,E1 17777.175,E2 17777.175} C_VEL
LIN {X 0,Y 437.354,Z 907.494,A -85,B 0,C 180,E1 17776.153,E2 17776.153} C_VEL
LIN {X 0,Y 431.428,Z 931.125,A -85,B 0,C 180,E1 17774.715,E2 17774.715} C_VEL
LIN {X 0,Y 426.09,Z 950.036,A -85,B 0,C 180,E1 17773.325,E2 17773.325} C_VEL
LIN {X 0,Y 419.765,Z 970.551,A -85,B 0,C 180,E1 17771.56,E2 17771.56} C_VEL
LIN {X 0,Y 413.292,Z 989.566,A -85,B 0,C 180,E1 17769.605,E2 17769.605} C_VEL
LIN {X 0,Y 406.705,Z 1008.039,A -85,B 0,C 180,E1 17767.391,E2 17767.391} C_VEL
LIN {X 0,Y 400.1,Z 1025.367,A -85,B 0,C 180,E1 17764.911,E2 17764.911} C_VEL
LIN {X 0,Y 393.851,Z 1041.533,A -85,B 0,C 180,E1 17762.218,E2 17762.218} C_VEL
LIN {X 0,Y 388.037,Z 1056.125,A -85,B 0,C 180,E1 17759.314,E2 17759.314} C_VEL
LIN {X 0,Y 382.853,Z 1069.577,A -85,B 0,C 180,E1 17756.192,E2 17756.192} C_VEL
LIN {X 0,Y 378.338,Z 1081.458,A -85,B 0,C 180,E1 17752.861,E2 17752.861} C_VEL
LIN {X 0,Y 374.792,Z 1091.694,A -85,B 0,C 180,E1 17749.48,E2 17749.48} C_VEL
LIN {X 0,Y 372.021,Z 1100.448,A -85,B 0,C 180,E1 17745.911,E2 17745.911} C_VEL
LIN {X 0,Y 370.193,Z 1107.367,A -85,B 0,C 180,E1 17742.479,E2 17742.479} C_VEL
LIN {X 0,Y 368.902,Z 1113.419,A -85,B 0,C 180,E1 17738.573,E2 17738.573} C_VEL
LIN {X 0,Y 368.344,Z 1117.158,A -85,B 0,C 180,E1 17735.296,E2 17735.296} C_VEL
LIN {X 0,Y 368.081,Z 1120.03,A -85,B 0,C 180,E1 17731.557,E2 17731.557} C_VEL
LIN {X 0,Y 368.019,Z 1121.199,A -85,B 0,C 180,E1 17728.132,E2 17728.132} C_VEL
LIN {X 0,Y 368.018,Z 1121.234,A -85,B 0,C 180,E1 17725.168,E2 17725.168} C_VEL
LIN {X 0,Y 368.125,Z 1120.263,A -85,B 0,C 180,E1 17722.037,E2 17722.037} C_VEL
LIN {X 0,Y 368.459,Z 1117.506,A -85,B 0,C 180,E1 17718.098,E2 17718.098} C_VEL
LIN {X 0,Y 369.135,Z 1113.833,A -85,B 0,C 180,E1 17714.767,E2 17714.767} C_VEL
LIN {X 0,Y 370.568,Z 1108.17,A -85,B 0,C 180,E1 17710.944,E2 17710.944} C_VEL
LIN {X 0,Y 372.761,Z 1100.937,A -85,B 0,C 180,E1 17707.278,E2 17707.278} C_VEL
LIN {X 0,Y 375.927,Z 1092.142,A -85,B 0,C 180,E1 17703.629,E2 17703.629} C_VEL
LIN {X 0,Y 379.932,Z 1081.779,A -85,B 0,C 180,E1 17700.171,E2 17700.171} C_VEL
LIN {X 0,Y 382.355,Z 1075.95,A -85,B 0,C 180,E1 17698.457,E2 17698.457} C_VEL
LIN {X 0,Y 382.946,Z 1072.464,A -85,B 0,C 180,E1 17697.422,E2 17697.422} C_VEL
LIN {X 0,Y 381.613,Z 1063.409,A -85,B 0,C 180,E1 17694.547,E2 17694.547} C_VEL
LIN {X 0,Y 382.472,Z 1059.991,A -85,B 0,C 180,E1 17693.7,E2 17693.7} C_VEL
LIN {X 0,Y 388.46,Z 1046.584,A -85,B 0,C 180,E1 17690.903,E2 17690.903} C_VEL
LIN {X 0,Y 395.433,Z 1031.011,A -85,B 0,C 180,E1 17688.122,E2 17688.122} C_VEL
LIN {X 0,Y 402.515,Z 1014.335,A -85,B 0,C 180,E1 17685.631,E2 17685.631} C_VEL
LIN {X 0,Y 409.827,Z 996.591,A -85,B 0,C 180,E1 17683.359,E2 17683.359} C_VEL
LIN {X 0,Y 417.184,Z 977.197,A -85,B 0,C 180,E1 17681.289,E2 17681.289} C_VEL
LIN {X 0,Y 423.997,Z 958.011,A -85,B 0,C 180,E1 17679.543,E2 17679.543} C_VEL
LIN {X 0,Y 430.662,Z 937.016,A -85,B 0,C 180,E1 17677.947,E2 17677.947} C_VEL
LIN {X 0,Y 436.364,Z 917.148,A -85,B 0,C 180,E1 17676.679,E2 17676.679} C_VEL
LIN {X 0,Y 442.298,Z 893.173,A -85,B 0,C 180,E1 17675.415,E2 17675.415} C_VEL
LIN {X 0,Y 446.645,Z 872.423,A -85,B 0,C 180,E1 17674.53,E2 17674.53} C_VEL
LIN {X 0,Y 450.957,Z 847.197,A -85,B 0,C 180,E1 17673.68,E2 17673.68} C_VEL
LIN {X 0,Y 453.799,Z 825.093,A -85,B 0,C 180,E1 17673.123,E2 17673.123} C_VEL
LIN {X 0,Y 456.086,Z 798.337,A -85,B 0,C 180,E1 17672.625,E2 17672.625} C_VEL
LIN {X 0,Y 470.277,Z 576.209,A -85,B 0,C 180,E1 17669.083,E2 17669.083} C_VEL
LIN {X 0,Y 461.755,Z 562.713,A -85,B 0,C 180,E1 17666.805,E2 17666.805} C_VEL
LIN {X 0,Y 452.926,Z 549.551,A -85,B 0,C 180,E1 17664.174,E2 17664.174} C_VEL
LIN {X 0,Y 445.371,Z 539.151,A -85,B 0,C 180,E1 17661.642,E2 17661.642} C_VEL
LIN {X 0,Y 441.028,Z 533.292,A -85,B 0,C 180,E1 17660.02,E2 17660.02} C_VEL
LIN {X 0,Y 438.103,Z 529.43,A -85,B 0,C 180,E1 17658.841,E2 17658.841} C_VEL
LIN {X 0,Y 434.363,Z 524.531,A -85,B 0,C 180,E1 17657.206,E2 17657.206} C_VEL
LIN {X 0,Y 430.557,Z 519.582,A -85,B 0,C 180,E1 17655.352,E2 17655.352} C_VEL
LIN {X 0,Y 427.039,Z 515,A -85,B 0,C 180,E1 17653.403,E2 17653.403} C_VEL
LIN {X 0,Y 425.282,Z 513.286,A -85,B 0,C 180,E1 17652.354,E2 17652.354} C_VEL
LIN {X 0,Y 422.457,Z 509.402,A -85,B 0,C 180,E1 17650.363,E2 17650.363} C_VEL
LIN {X 0,Y 421.792,Z 508.357,A -85,B 0,C 180,E1 17649.828,E2 17649.828} C_VEL
LIN {X 0,Y 418.859,Z 505.725,A -85,B 0,C 180,E1 17647.269,E2 17647.269} C_VEL
LIN {X 0,Y 417.188,Z 502.354,A -85,B 0,C 180,E1 17645.088,E2 17645.088} C_VEL
LIN {X 0,Y 414.778,Z 501.013,A -85,B 0,C 180,E1 17638.757,E2 17638.757} C_VEL
LIN {X 0,Y 417.154,Z 502.308,A -85,B 0,C 180,E1 17632.425,E2 17632.425} C_VEL
LIN {X 0,Y 419.772,Z 506.807,A -85,B 0,C 180,E1 17629.292,E2 17629.292} C_VEL
LIN {X 0,Y 422.25,Z 508.921,A -85,B 0,C 180,E1 17627.278,E2 17627.278} C_VEL
LIN {X 0,Y 425.013,Z 512.971,A -85,B 0,C 180,E1 17625.281,E2 17625.281} C_VEL
LIN {X 0,Y 426.975,Z 514.915,A -85,B 0,C 180,E1 17624.098,E2 17624.098} C_VEL
LIN {X 0,Y 430.49,Z 519.489,A -85,B 0,C 180,E1 17622.146,E2 17622.146} C_VEL
LIN {X 0,Y 433.942,Z 524.075,A -85,B 0,C 180,E1 17620.447,E2 17620.447} C_VEL
LIN {X 0,Y 438.251,Z 530.532,A -85,B 0,C 180,E1 17618.519,E2 17618.519} C_VEL
LIN {X 0,Y 443.569,Z 538.333,A -85,B 0,C 180,E1 17616.414,E2 17616.414} C_VEL
LIN {X 0,Y 452.208,Z 551.967,A -85,B 0,C 180,E1 17613.4,E2 17613.4} C_VEL
LIN {X 0,Y 461.524,Z 567.684,A -85,B 0,C 180,E1 17610.561,E2 17610.561} C_VEL
LIN {X 0,Y 469.712,Z 582.67,A -85,B 0,C 180,E1 17608.314,E2 17608.314} C_VEL
LIN {X 0,Y 470.027,Z 583.823,A -85,B 0,C 180,E1 17608.215,E2 17608.215} C_VEL
LIN {X 0,Y 456.231,Z 800.934,A -85,B 0,C 180,E1 17604.738,E2 17604.738} C_VEL
LIN {X 0,Y 453.531,Z 838.587,A -85,B 0,C 180,E1 17604.098,E2 17604.098} C_VEL
LIN {X 0,Y 450.476,Z 862.153,A -85,B 0,C 180,E1 17603.559,E2 17603.559} C_VEL
LIN {X 0,Y 446.384,Z 886.26,A -85,B 0,C 180,E1 17602.844,E2 17602.844} C_VEL
LIN {X 0,Y 441.358,Z 909.538,A -85,B 0,C 180,E1 17601.93,E2 17601.93} C_VEL
LIN {X 0,Y 435.835,Z 931.878,A -85,B 0,C 180,E1 17600.845,E2 17600.845} C_VEL
LIN {X 0,Y 429.376,Z 954.251,A -85,B 0,C 180,E1 17599.493,E2 17599.493} C_VEL
LIN {X 0,Y 422.926,Z 974.503,A -85,B 0,C 180,E1 17598.035,E2 17598.035} C_VEL
LIN {X 0,Y 415.542,Z 995.502,A -85,B 0,C 180,E1 17596.209,E2 17596.209} C_VEL
LIN {X 0,Y 408.827,Z 1013.308,A -85,B 0,C 180,E1 17594.386,E2 17594.386} C_VEL
LIN {X 0,Y 400.835,Z 1033.292,A -85,B 0,C 180,E1 17591.954,E2 17591.954} C_VEL
LIN {X 0,Y 394.332,Z 1048.878,A -85,B 0,C 180,E1 17589.716,E2 17589.716} C_VEL
LIN {X 0,Y 386.842,Z 1066.434,A -85,B 0,C 180,E1 17586.748,E2 17586.748} C_VEL
LIN {X 0,Y 380.946,Z 1080.178,A -85,B 0,C 180,E1 17583.992,E2 17583.992} C_VEL
LIN {X 0,Y 374.974,Z 1094.468,A -85,B 0,C 180,E1 17580.618,E2 17580.618} C_VEL
LIN {X 0,Y 370.501,Z 1105.604,A -85,B 0,C 180,E1 17577.483,E2 17577.483} C_VEL
LIN {X 0,Y 366.63,Z 1116.237,A -85,B 0,C 180,E1 17573.976,E2 17573.976} C_VEL
LIN {X 0,Y 363.668,Z 1125.35,A -85,B 0,C 180,E1 17570.269,E2 17570.269} C_VEL
LIN {X 0,Y 361.705,Z 1132.907,A -85,B 0,C 180,E1 17566.543,E2 17566.543} C_VEL
LIN {X 0,Y 360.534,Z 1138.934,A -85,B 0,C 180,E1 17562.656,E2 17562.656} C_VEL
LIN {X 0,Y 360.098,Z 1142.714,A -85,B 0,C 180,E1 17559.429,E2 17559.429} C_VEL
LIN {X 0,Y 359.976,Z 1145.728,A -85,B 0,C 180,E1 17555.739,E2 17555.739} C_VEL
LIN {X 0,Y 360.014,Z 1147.083,A -85,B 0,C 180,E1 17552.069,E2 17552.069} C_VEL
